Yaskawa INFORM job: Cilinder_ROBODK.jbi

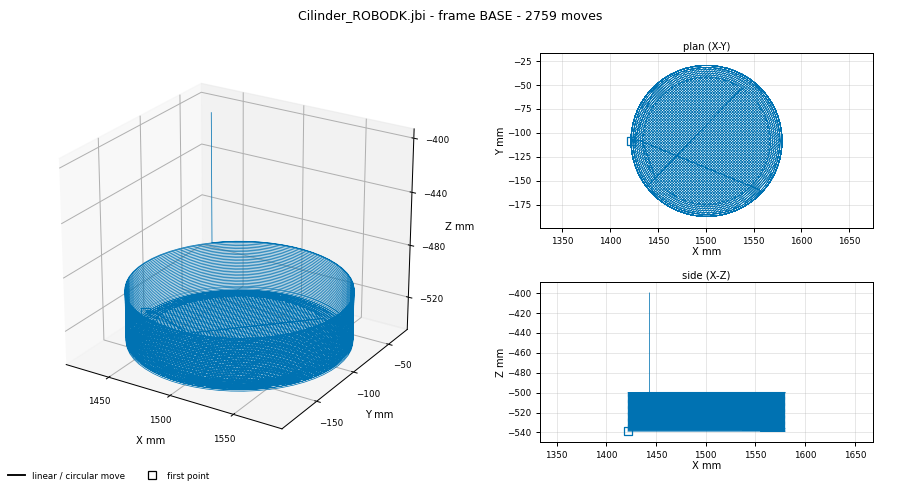
[picture p0: tool path of Cilinder_ROBODK.jbi in frame BASE, 2759 of 2760 moves have a stored position in this frame; points joined in program order, loops and branches not executed]
/JOB
//NAME CILINDER
//POS
///NPOS 2760,0,0,0,0,0
///TOOL 9
///POSTYPE PULSE
///PULSE
C00000=-4,42,-29,0,-18,-176
///TOOL 9
///POSTYPE BASE
///RECTAN
///RCONF 0,0,0,0,0,0,0,0
C00001=1421.799,-108.483,-538.800,180.00,-0.00,180.00
C00002=1422.262,-99.945,-538.800,180.00,0.00,-180.00
C00003=1423.646,-91.503,-538.800,180.00,-0.00,180.00
C00004=1425.931,-83.274,-538.800,180.00,-0.00,-180.00
C00005=1429.100,-75.315,-538.800,180.00,0.00,-180.00
C00006=1433.106,-67.758,-538.800,180.00,0.00,180.00
C00007=1437.906,-60.678,-538.800,180.00,-0.00,-180.00
C00008=1443.445,-54.158,-538.800,180.00,-0.00,-180.00
C00009=1449.655,-48.276,-538.800,180.00,0.00,180.00
C00010=1456.467,-43.098,-538.800,180.00,-0.00,-180.00
C00011=1463.794,-38.689,-538.800,180.00,-0.00,-180.00
C00012=1471.559,-35.097,-538.800,180.00,0.00,180.00
C00013=1479.661,-32.366,-538.800,180.00,0.00,-180.00
C00014=1488.017,-30.527,-538.800,180.00,0.00,180.00
C00015=1496.522,-29.601,-538.800,180.00,-0.00,180.00
C00016=1505.072,-29.601,-538.800,180.00,-0.00,-180.00
C00017=1513.577,-30.527,-538.800,180.00,-0.00,-180.00
C00018=1521.933,-32.366,-538.800,180.00,-0.00,-180.00
C00019=1530.035,-35.097,-538.800,180.00,0.00,180.00
C00020=1537.800,-38.689,-538.800,180.00,0.00,-180.00
C00021=1545.127,-43.098,-538.800,180.00,0.00,180.00
C00022=1551.939,-48.276,-538.800,180.00,0.00,-180.00
C00023=1558.149,-54.158,-538.800,180.00,0.00,-180.00
C00024=1563.688,-60.678,-538.800,180.00,-0.00,-180.00
C00025=1568.488,-67.758,-538.800,180.00,-0.00,180.00
C00026=1572.494,-75.315,-538.800,180.00,0.00,-180.00
C00027=1575.665,-83.274,-538.800,180.00,0.00,180.00
C00028=1577.948,-91.503,-538.800,180.00,0.00,-180.00
C00029=1579.332,-99.945,-538.800,180.00,-0.00,180.00
C00030=1579.795,-108.486,-538.800,180.00,0.00,-180.00
C00031=1579.332,-117.025,-538.800,180.00,0.00,-180.00
C00032=1577.948,-125.467,-538.800,180.00,-0.00,-180.00
C00033=1575.663,-133.694,-538.800,180.00,-0.00,-180.00
C00034=1572.494,-141.653,-538.800,180.00,-0.00,-180.00
C00035=1568.486,-149.212,-538.800,180.00,0.00,-180.00
C00036=1563.686,-156.292,-538.800,180.00,0.00,-180.00
C00037=1558.149,-162.810,-538.800,180.00,0.00,-180.00
C00038=1551.937,-168.694,-538.800,180.00,0.00,-180.00
C00039=1545.128,-173.870,-538.800,180.00,-0.00,-180.00
C00040=1537.800,-178.279,-538.800,180.00,-0.00,-180.00
C00041=1530.035,-181.871,-538.800,180.00,0.00,-180.00
C00042=1521.933,-184.602,-538.800,180.00,0.00,180.00
C00043=1513.577,-186.441,-538.800,180.00,0.00,-180.00
C00044=1505.072,-187.366,-538.800,180.00,0.00,-180.00
C00045=1496.522,-187.366,-538.800,180.00,0.00,180.00
C00046=1488.017,-186.441,-538.800,180.00,-0.00,-180.00
C00047=1479.661,-184.602,-538.800,180.00,-0.00,-180.00
C00048=1471.559,-181.871,-538.800,180.00,-0.00,-180.00
C00049=1463.794,-178.279,-538.800,180.00,-0.00,-180.00
C00050=1456.467,-173.870,-538.800,180.00,0.00,-180.00
C00051=1449.655,-168.692,-538.800,180.00,0.00,-180.00
C00052=1443.445,-162.810,-538.800,180.00,-0.00,-180.00
C00053=1437.906,-156.290,-538.800,180.00,0.00,-180.00
C00054=1433.106,-149.210,-538.800,180.00,0.00,-180.00
C00055=1429.100,-141.653,-538.800,180.00,0.00,180.00
C00056=1425.929,-133.694,-538.800,180.00,0.00,-180.00
C00057=1423.646,-125.465,-538.800,180.00,0.00,-180.00
C00058=1422.262,-117.023,-538.800,180.00,0.00,-180.00
C00059=1421.799,-108.483,-538.800,180.00,-0.00,180.00
C00060=1421.846,-107.610,-538.800,180.00,-0.00,-180.00
C00061=1424.567,-107.757,-538.800,180.00,0.00,-180.00
C00062=1424.528,-108.484,-538.800,180.00,-0.00,-180.00
C00063=1423.702,-108.482,-538.800,180.00,0.00,-180.00
C00064=1424.154,-100.153,-538.800,180.00,-0.00,180.00
C00065=1425.505,-91.912,-538.800,180.00,-0.00,-180.00
C00066=1427.735,-83.882,-538.800,180.00,0.00,-180.00
C00067=1430.827,-76.115,-538.800,180.00,0.00,-180.00
C00068=1434.736,-68.740,-538.800,180.00,-0.00,-180.00
C00069=1439.419,-61.831,-538.800,180.00,-0.00,-180.00
C00070=1444.826,-55.468,-538.800,180.00,0.00,-180.00
C00071=1450.887,-49.728,-538.800,180.00,-0.00,180.00
C00072=1457.537,-44.673,-538.800,180.00,0.00,-180.00
C00073=1464.686,-40.372,-538.800,180.00,-0.00,-180.00
C00074=1472.266,-36.865,-538.800,180.00,-0.00,-180.00
C00075=1480.169,-34.201,-538.800,180.00,0.00,-180.00
C00076=1488.326,-32.405,-538.800,180.00,0.00,-180.00
C00077=1496.627,-31.501,-538.800,180.00,-0.00,180.00
C00078=1504.967,-31.501,-538.800,180.00,0.00,-180.00
C00079=1513.268,-32.405,-538.800,180.00,0.00,-180.00
C00080=1521.425,-34.201,-538.800,180.00,0.00,-180.00
C00081=1529.328,-36.865,-538.800,180.00,-0.00,180.00
C00082=1536.908,-40.372,-538.800,180.00,-0.00,-180.00
C00083=1544.056,-44.673,-538.800,180.00,-0.00,180.00
C00084=1550.707,-49.728,-538.800,180.00,0.00,180.00
C00085=1556.768,-55.468,-538.800,180.00,0.00,-180.00
C00086=1562.175,-61.831,-538.800,180.00,-0.00,-180.00
C00087=1566.858,-68.740,-538.800,180.00,-0.00,-180.00
C00088=1570.767,-76.115,-538.800,180.00,-0.00,-180.00
C00089=1573.867,-83.896,-538.800,180.00,0.00,180.00
C00090=1576.089,-91.913,-538.800,180.00,-0.00,-180.00
C00091=1577.440,-100.153,-538.800,180.00,-0.00,-180.00
C00092=1577.892,-108.487,-538.800,180.00,0.00,-180.00
C00093=1577.440,-116.819,-538.800,180.00,-0.00,-180.00
C00094=1576.089,-125.059,-538.800,180.00,0.00,-180.00
C00095=1573.863,-133.072,-538.800,180.00,-0.00,180.00
C00096=1570.766,-140.853,-538.800,180.00,-0.00,-180.00
C00097=1566.854,-148.232,-538.800,180.00,-0.00,-180.00
C00098=1562.172,-155.139,-538.800,180.00,-0.00,-180.00
C00099=1556.768,-161.501,-538.800,180.00,0.00,-180.00
C00100=1550.703,-167.244,-538.800,180.00,-0.00,180.00
C00101=1544.058,-172.295,-538.800,180.00,-0.00,-180.00
C00102=1536.908,-176.596,-538.800,180.00,0.00,-180.00
C00103=1529.328,-180.103,-538.800,180.00,0.00,-180.00
C00104=1521.425,-182.767,-538.800,180.00,-0.00,180.00
C00105=1513.268,-184.563,-538.800,180.00,-0.00,-180.00
C00106=1504.967,-185.465,-538.800,180.00,-0.00,180.00
C00107=1496.627,-185.466,-538.800,180.00,-0.00,-180.00
C00108=1488.326,-184.563,-538.800,180.00,-0.00,180.00
C00109=1480.169,-182.767,-538.800,180.00,-0.00,-180.00
C00110=1472.266,-180.103,-538.800,180.00,0.00,-180.00
C00111=1464.686,-176.596,-538.800,180.00,0.00,-180.00
C00112=1457.537,-172.295,-538.800,180.00,0.00,-180.00
C00113=1450.887,-167.240,-538.800,180.00,0.00,180.00
C00114=1444.826,-161.500,-538.800,180.00,0.00,-180.00
C00115=1439.419,-155.137,-538.800,180.00,0.00,180.00
C00116=1434.736,-148.228,-538.800,180.00,0.00,-180.00
C00117=1430.827,-140.853,-538.800,180.00,0.00,180.00
C00118=1427.727,-133.072,-538.800,180.00,0.00,-180.00
C00119=1425.505,-125.055,-538.800,180.00,0.00,180.00
C00120=1424.154,-116.815,-538.800,180.00,0.00,-180.00
C00121=1423.702,-108.482,-538.800,180.00,0.00,-180.00
C00122=1424.528,-108.484,-538.800,180.00,-0.00,-180.00
C00123=1445.040,-56.761,-538.800,180.00,-0.00,180.00
C00124=1447.262,-54.539,-538.800,180.00,0.00,-180.00
C00125=1460.678,-43.951,-538.800,180.00,0.00,180.00
C00126=1436.060,-68.569,-538.800,180.00,-0.00,180.00
C00127=1435.707,-68.922,-538.800,180.00,0.00,-180.00
C00128=1432.654,-74.803,-538.800,180.00,0.00,-180.00
C00129=1467.099,-40.359,-538.800,180.00,0.00,-180.00
C00130=1467.452,-40.006,-538.800,180.00,-0.00,-180.00
C00131=1472.362,-37.924,-538.800,180.00,0.00,-180.00
C00132=1430.403,-79.883,-538.800,180.00,0.00,180.00
C00133=1430.050,-80.236,-538.800,180.00,-0.00,-180.00
C00134=1430.069,-80.243,-538.800,180.00,0.00,-180.00
C00135=1428.596,-84.518,-538.800,180.00,-0.00,-180.00
C00136=1476.681,-36.433,-538.800,180.00,0.00,180.00
C00137=1477.034,-36.080,-538.800,180.00,-0.00,-180.00
C00138=1477.047,-36.120,-538.800,180.00,-0.00,180.00
C00139=1480.871,-35.072,-538.800,180.00,0.00,-180.00
C00140=1427.508,-88.435,-538.800,180.00,0.00,-180.00
C00141=1427.155,-88.788,-538.800,180.00,0.00,-180.00
C00142=1427.222,-88.805,-538.800,180.00,0.00,-180.00
C00143=1426.450,-92.321,-538.800,180.00,-0.00,-180.00
C00144=1484.499,-34.273,-538.800,180.00,0.00,-180.00
C00145=1488.126,-33.474,-538.800,180.00,-0.00,180.00
C00146=1425.896,-95.704,-538.800,180.00,0.00,-180.00
C00147=1425.341,-99.087,-538.800,180.00,-0.00,180.00
C00148=1491.345,-33.083,-538.800,180.00,0.00,-180.00
C00149=1494.519,-32.738,-538.800,180.00,0.00,-180.00
C00150=1425.043,-102.214,-538.800,180.00,0.00,-180.00
C00151=1424.880,-105.205,-538.800,180.00,0.00,-180.00
C00152=1497.583,-32.502,-538.800,180.00,0.00,-180.00
C00153=1500.411,-32.502,-538.800,180.00,0.00,180.00
C00154=1424.718,-108.195,-538.800,180.00,0.00,-180.00
C00155=1424.834,-110.908,-538.800,180.00,0.00,180.00
C00156=1503.240,-32.502,-538.800,180.00,0.00,-180.00
C00157=1505.954,-32.616,-538.800,180.00,0.00,-180.00
C00158=1424.980,-113.590,-538.800,180.00,-0.00,180.00
C00159=1425.126,-116.273,-538.800,180.00,-0.00,-180.00
C00160=1508.505,-32.894,-538.800,180.00,0.00,180.00
C00161=1511.055,-33.172,-538.800,180.00,0.00,-180.00
C00162=1425.483,-118.744,-538.800,180.00,-0.00,180.00
C00163=1425.882,-121.174,-538.800,180.00,-0.00,-180.00
C00164=1513.561,-33.495,-538.800,180.00,-0.00,180.00
C00165=1515.879,-34.005,-538.800,180.00,-0.00,180.00
C00166=1426.280,-123.604,-538.800,180.00,0.00,-180.00
C00167=1426.784,-125.929,-538.800,180.00,-0.00,-180.00
C00168=1518.196,-34.516,-538.800,180.00,-0.00,180.00
C00169=1520.514,-35.027,-538.800,180.00,0.00,180.00
C00170=1427.398,-128.143,-538.800,180.00,-0.00,-180.00
C00171=1428.011,-130.358,-538.800,180.00,-0.00,180.00
C00172=1522.686,-35.683,-538.800,180.00,-0.00,180.00
C00173=1524.802,-36.396,-538.800,180.00,-0.00,180.00
C00174=1428.625,-132.573,-538.800,180.00,-0.00,-180.00
C00175=1429.415,-134.611,-538.800,180.00,0.00,-180.00
C00176=1526.917,-37.109,-538.800,180.00,-0.00,-180.00
C00177=1529.026,-37.829,-538.800,180.00,-0.00,180.00
C00178=1430.221,-136.634,-538.800,180.00,0.00,-180.00
C00179=1431.026,-138.657,-538.800,180.00,-0.00,180.00
C00180=1530.960,-38.723,-538.800,180.00,0.00,-180.00
C00181=1532.893,-39.619,-538.800,180.00,0.00,180.00
C00182=1431.853,-140.658,-538.800,180.00,-0.00,180.00
C00183=1432.833,-142.507,-538.800,180.00,0.00,180.00
C00184=1534.827,-40.513,-538.800,180.00,-0.00,-180.00
C00185=1536.733,-41.436,-538.800,180.00,0.00,-180.00
C00186=1433.812,-144.356,-538.800,180.00,-0.00,-180.00
C00187=1434.792,-146.204,-538.800,180.00,0.00,-180.00
C00188=1538.499,-42.498,-538.800,180.00,0.00,180.00
C00189=1540.265,-43.561,-538.800,180.00,0.00,-180.00
C00190=1435.802,-148.023,-538.800,180.00,0.00,-180.00
C00191=1436.945,-149.709,-538.800,180.00,0.00,-180.00
C00192=1542.030,-44.623,-538.800,180.00,0.00,-180.00
C00193=1543.769,-45.713,-538.800,180.00,0.00,180.00
C00194=1438.088,-151.394,-538.800,180.00,-0.00,-180.00
C00195=1439.230,-153.080,-538.800,180.00,0.00,-180.00
C00196=1545.376,-46.934,-538.800,180.00,-0.00,-180.00
C00197=1546.983,-48.155,-538.800,180.00,-0.00,-180.00
C00198=1440.395,-154.744,-538.800,180.00,0.00,-180.00
C00199=1441.695,-156.273,-538.800,180.00,0.00,-180.00
C00200=1548.590,-49.377,-538.800,180.00,-0.00,-180.00
C00201=1550.184,-50.612,-538.800,180.00,-0.00,180.00
C00202=1442.994,-157.802,-538.800,180.00,0.00,180.00
C00203=1444.293,-159.331,-538.800,180.00,0.00,-180.00
C00204=1551.636,-51.988,-538.800,180.00,0.00,-180.00
C00205=1553.089,-53.363,-538.800,180.00,-0.00,-180.00
C00206=1445.598,-160.855,-538.800,180.00,-0.00,-180.00
C00207=1447.051,-162.230,-538.800,180.00,-0.00,180.00
C00208=1554.542,-54.739,-538.800,180.00,0.00,180.00
C00209=1555.994,-56.115,-538.800,180.00,-0.00,-180.00
C00210=1448.503,-163.606,-538.800,180.00,0.00,-180.00
C00211=1449.956,-164.982,-538.800,180.00,0.00,-180.00
C00212=1557.299,-57.639,-538.800,180.00,0.00,-180.00
C00213=1558.598,-59.168,-538.800,180.00,-0.00,-180.00
C00214=1451.409,-166.357,-538.800,180.00,0.00,-180.00
C00215=1453.002,-167.593,-538.800,180.00,0.00,180.00
C00216=1559.898,-60.697,-538.800,180.00,-0.00,-180.00
C00217=1561.198,-62.225,-538.800,180.00,-0.00,-180.00
C00218=1454.609,-168.814,-538.800,180.00,0.00,-180.00
C00219=1456.216,-170.036,-538.800,180.00,0.00,-180.00
C00220=1562.362,-63.889,-538.800,180.00,0.00,-180.00
C00221=1563.504,-65.576,-538.800,180.00,-0.00,180.00
C00222=1457.823,-171.257,-538.800,180.00,-0.00,180.00
C00223=1459.562,-172.347,-538.800,180.00,-0.00,180.00
C00224=1564.647,-67.261,-538.800,180.00,0.00,-180.00
C00225=1565.790,-68.947,-538.800,180.00,-0.00,180.00
C00226=1461.328,-173.409,-538.800,180.00,-0.00,-180.00
C00227=1463.094,-174.472,-538.800,180.00,-0.00,180.00
C00228=1566.799,-70.766,-538.800,180.00,-0.00,-180.00
C00229=1567.779,-72.614,-538.800,180.00,0.00,180.00
C00230=1464.860,-175.534,-538.800,180.00,-0.00,180.00
C00231=1466.766,-176.456,-538.800,180.00,0.00,-180.00
C00232=1568.759,-74.463,-538.800,180.00,-0.00,-180.00
C00233=1569.739,-76.312,-538.800,180.00,-0.00,-180.00
C00234=1468.699,-177.352,-538.800,180.00,0.00,-180.00
C00235=1470.633,-178.246,-538.800,180.00,0.00,180.00
C00236=1570.565,-78.314,-538.800,180.00,0.00,-180.00
C00237=1571.372,-80.336,-538.800,180.00,-0.00,-180.00
C00238=1472.566,-179.141,-538.800,180.00,-0.00,-180.00
C00239=1474.675,-179.860,-538.800,180.00,0.00,-180.00
C00240=1572.178,-82.358,-538.800,180.00,0.00,180.00
C00241=1572.968,-84.397,-538.800,180.00,0.00,180.00
C00242=1476.791,-180.573,-538.800,180.00,-0.00,180.00
C00243=1478.906,-181.287,-538.800,180.00,0.00,-180.00
C00244=1573.581,-86.611,-538.800,180.00,0.00,-180.00
C00245=1574.195,-88.826,-538.800,180.00,0.00,-180.00
C00246=1481.078,-181.944,-538.800,180.00,0.00,-180.00
C00247=1483.395,-182.454,-538.800,180.00,-0.00,-180.00
C00248=1574.809,-91.041,-538.800,180.00,-0.00,-180.00
C00249=1575.313,-93.365,-538.800,180.00,0.00,-180.00
C00250=1485.713,-182.965,-538.800,180.00,0.00,-180.00
C00251=1488.031,-183.475,-538.800,180.00,0.00,-180.00
C00252=1575.711,-95.795,-538.800,180.00,0.00,-180.00
C00253=1576.109,-98.226,-538.800,180.00,-0.00,180.00
C00254=1490.537,-183.798,-538.800,180.00,-0.00,-180.00
C00255=1493.088,-184.075,-538.800,180.00,0.00,180.00
C00256=1576.466,-100.697,-538.800,180.00,-0.00,180.00
C00257=1576.612,-103.380,-538.800,180.00,0.00,-180.00
C00258=1495.639,-184.353,-538.800,180.00,-0.00,-180.00
C00259=1498.354,-184.466,-538.800,180.00,0.00,180.00
C00260=1576.758,-106.062,-538.800,180.00,0.00,180.00
C00261=1576.874,-108.774,-538.800,180.00,0.00,-180.00
C00262=1501.183,-184.466,-538.800,180.00,0.00,180.00
C00263=1504.011,-184.466,-538.800,180.00,0.00,-180.00
C00264=1576.712,-111.765,-538.800,180.00,-0.00,-180.00
C00265=1576.549,-114.756,-538.800,180.00,0.00,-180.00
C00266=1507.075,-184.230,-538.800,180.00,-0.00,180.00
C00267=1510.248,-183.886,-538.800,180.00,0.00,-180.00
C00268=1576.251,-117.883,-538.800,180.00,0.00,180.00
C00269=1575.696,-121.266,-538.800,180.00,-0.00,-180.00
C00270=1513.467,-183.496,-538.800,180.00,-0.00,-180.00
C00271=1517.093,-182.697,-538.800,180.00,0.00,180.00
C00272=1575.143,-124.648,-538.800,180.00,0.00,-180.00
C00273=1575.496,-124.295,-538.800,180.00,0.00,-180.00
C00274=1575.383,-124.277,-538.800,180.00,-0.00,180.00
C00275=1574.085,-128.534,-538.800,180.00,0.00,-180.00
C00276=1520.721,-181.898,-538.800,180.00,-0.00,180.00
C00277=1520.368,-182.251,-538.800,180.00,0.00,-180.00
C00278=1520.348,-182.163,-538.800,180.00,-0.00,-180.00
C00279=1524.911,-180.536,-538.800,180.00,-0.00,-180.00
C00280=1572.997,-132.450,-538.800,180.00,0.00,180.00
C00281=1573.350,-132.097,-538.800,180.00,0.00,-180.00
C00282=1573.284,-132.080,-538.800,180.00,0.00,-180.00
C00283=1571.188,-137.088,-538.800,180.00,0.00,-180.00
C00284=1529.230,-179.046,-538.800,180.00,-0.00,180.00
C00285=1528.877,-179.399,-538.800,180.00,0.00,-180.00
C00286=1528.874,-179.390,-538.800,180.00,-0.00,-180.00
C00287=1534.493,-176.611,-538.800,180.00,-0.00,180.00
C00288=1568.937,-142.167,-538.800,180.00,0.00,-180.00
C00289=1569.290,-141.814,-538.800,180.00,0.00,-180.00
C00290=1565.528,-148.405,-538.800,180.00,0.00,-180.00
C00291=1540.914,-173.018,-538.800,180.00,-0.00,180.00
C00292=1540.561,-173.371,-538.800,180.00,-0.00,-180.00
C00293=1554.330,-162.432,-538.800,180.00,0.00,-180.00
C00294=1556.551,-160.211,-538.800,180.00,-0.00,180.00
C00295=1555.237,-159.097,-538.800,180.00,0.00,180.00
C00296=1555.237,-159.097,-537.600,180.00,0.00,180.00
C00297=1431.814,-108.483,-537.600,180.00,-0.00,180.00
C00298=1432.218,-101.027,-537.600,180.00,0.00,-180.00
C00299=1433.426,-93.656,-537.600,180.00,-0.00,-180.00
C00300=1435.421,-86.471,-537.600,180.00,-0.00,-180.00
C00301=1438.190,-79.519,-537.600,180.00,0.00,-180.00
C00302=1441.687,-72.920,-537.600,180.00,0.00,180.00
C00303=1445.878,-66.739,-537.600,180.00,-0.00,-180.00
C00304=1450.715,-61.046,-537.600,180.00,-0.00,180.00
C00305=1456.138,-55.909,-537.600,180.00,0.00,-180.00
C00306=1462.087,-51.388,-537.600,180.00,0.00,-180.00
C00307=1468.485,-47.537,-537.600,180.00,0.00,-180.00
C00308=1475.266,-44.400,-537.600,180.00,0.00,-180.00
C00309=1482.341,-42.016,-537.600,180.00,-0.00,180.00
C00310=1489.637,-40.409,-537.600,180.00,0.00,-180.00
C00311=1497.064,-39.601,-537.600,180.00,-0.00,-180.00
C00312=1504.530,-39.601,-537.600,180.00,0.00,-180.00
C00313=1511.957,-40.409,-537.600,180.00,0.00,-180.00
C00314=1519.253,-42.016,-537.600,180.00,0.00,-180.00
C00315=1526.328,-44.400,-537.600,180.00,-0.00,180.00
C00316=1533.109,-47.537,-537.600,180.00,0.00,-180.00
C00317=1539.507,-51.387,-537.600,180.00,-0.00,180.00
C00318=1545.456,-55.909,-537.600,180.00,0.00,-180.00
C00319=1550.879,-61.046,-537.600,180.00,0.00,-180.00
C00320=1555.716,-66.739,-537.600,180.00,0.00,180.00
C00321=1559.907,-72.920,-537.600,180.00,0.00,180.00
C00322=1563.404,-79.520,-537.600,180.00,-0.00,-180.00
C00323=1566.175,-86.471,-537.600,180.00,-0.00,-180.00
C00324=1568.167,-93.654,-537.600,180.00,0.00,180.00
C00325=1569.376,-101.027,-537.600,180.00,0.00,180.00
C00326=1569.780,-108.486,-537.600,180.00,-0.00,180.00
C00327=1569.376,-115.943,-537.600,180.00,-0.00,-180.00
C00328=1568.168,-123.314,-537.600,180.00,0.00,-180.00
C00329=1566.173,-130.496,-537.600,180.00,0.00,180.00
C00330=1563.404,-137.449,-537.600,180.00,0.00,180.00
C00331=1559.905,-144.049,-537.600,180.00,0.00,180.00
C00332=1555.714,-150.232,-537.600,180.00,-0.00,-180.00
C00333=1550.879,-155.922,-537.600,180.00,-0.00,-180.00
C00334=1545.454,-161.061,-537.600,180.00,-0.00,-180.00
C00335=1539.508,-165.580,-537.600,180.00,-0.00,-180.00
C00336=1533.109,-169.430,-537.600,180.00,0.00,-180.00
C00337=1526.328,-172.568,-537.600,180.00,-0.00,180.00
C00338=1519.253,-174.952,-537.600,180.00,-0.00,-180.00
C00339=1511.957,-176.558,-537.600,180.00,0.00,-180.00
C00340=1504.530,-177.366,-537.600,180.00,0.00,-180.00
C00341=1497.064,-177.366,-537.600,180.00,0.00,180.00
C00342=1489.637,-176.558,-537.600,180.00,-0.00,180.00
C00343=1482.341,-174.952,-537.600,180.00,-0.00,-180.00
C00344=1475.266,-172.568,-537.600,180.00,0.00,-180.00
C00345=1468.485,-169.431,-537.600,180.00,0.00,180.00
C00346=1462.087,-165.581,-537.600,180.00,0.00,180.00
C00347=1456.138,-161.059,-537.600,180.00,-0.00,-180.00
C00348=1450.715,-155.922,-537.600,180.00,-0.00,180.00
C00349=1445.878,-150.229,-537.600,180.00,0.00,180.00
C00350=1441.687,-144.048,-537.600,180.00,0.00,-180.00
C00351=1438.190,-137.448,-537.600,180.00,0.00,-180.00
C00352=1435.419,-130.497,-537.600,180.00,-0.00,-180.00
C00353=1433.426,-123.314,-537.600,180.00,-0.00,-180.00
C00354=1432.218,-115.941,-537.600,180.00,-0.00,180.00
C00355=1431.814,-108.483,-537.600,180.00,-0.00,180.00
C00356=1429.811,-108.483,-537.600,180.00,-0.00,-180.00
C00357=1430.227,-100.811,-537.600,180.00,-0.00,-180.00
C00358=1431.470,-93.225,-537.600,180.00,-0.00,-180.00
C00359=1433.523,-85.832,-537.600,180.00,-0.00,-180.00
C00360=1436.372,-78.678,-537.600,180.00,0.00,-180.00
C00361=1439.971,-71.888,-537.600,180.00,0.00,-180.00
C00362=1444.284,-65.526,-537.600,180.00,0.00,-180.00
C00363=1449.261,-59.668,-537.600,180.00,-0.00,-180.00
C00364=1454.841,-54.382,-537.600,180.00,0.00,180.00
C00365=1460.963,-49.730,-537.600,180.00,-0.00,180.00
C00366=1467.547,-45.768,-537.600,180.00,0.00,-180.00
C00367=1474.525,-42.540,-537.600,180.00,-0.00,-180.00
C00368=1481.805,-40.086,-537.600,180.00,0.00,-180.00
C00369=1489.313,-38.433,-537.600,180.00,-0.00,-180.00
C00370=1496.956,-37.601,-537.600,180.00,0.00,-180.00
C00371=1504.638,-37.601,-537.600,180.00,-0.00,180.00
C00372=1512.281,-38.433,-537.600,180.00,0.00,-180.00
C00373=1519.789,-40.086,-537.600,180.00,0.00,180.00
C00374=1527.069,-42.540,-537.600,180.00,-0.00,-180.00
C00375=1534.047,-45.768,-537.600,180.00,0.00,180.00
C00376=1540.631,-49.730,-537.600,180.00,-0.00,180.00
C00377=1546.753,-54.382,-537.600,180.00,-0.00,-180.00
C00378=1552.333,-59.668,-537.600,180.00,-0.00,-180.00
C00379=1557.310,-65.526,-537.600,180.00,-0.00,180.00
C00380=1561.623,-71.888,-537.600,180.00,0.00,-180.00
C00381=1565.222,-78.679,-537.600,180.00,-0.00,-180.00
C00382=1568.073,-85.832,-537.600,180.00,0.00,-180.00
C00383=1570.124,-93.224,-537.600,180.00,0.00,180.00
C00384=1571.367,-100.811,-537.600,180.00,0.00,-180.00
C00385=1571.783,-108.486,-537.600,180.00,0.00,-180.00
C00386=1571.367,-116.159,-537.600,180.00,-0.00,-180.00
C00387=1570.124,-123.745,-537.600,180.00,-0.00,-180.00
C00388=1568.071,-131.136,-537.600,180.00,0.00,-180.00
C00389=1565.222,-138.290,-537.600,180.00,-0.00,-180.00
C00390=1561.621,-145.082,-537.600,180.00,-0.00,-180.00
C00391=1557.308,-151.444,-537.600,180.00,-0.00,180.00
C00392=1552.333,-157.300,-537.600,180.00,0.00,180.00
C00393=1546.751,-162.588,-537.600,180.00,0.00,-180.00
C00394=1540.632,-167.238,-537.600,180.00,0.00,-180.00
C00395=1534.048,-171.200,-537.600,180.00,-0.00,-180.00
C00396=1527.069,-174.428,-537.600,180.00,0.00,180.00
C00397=1519.789,-176.882,-537.600,180.00,0.00,180.00
C00398=1512.281,-178.535,-537.600,180.00,0.00,-180.00
C00399=1504.638,-179.366,-537.600,180.00,0.00,-180.00
C00400=1496.956,-179.366,-537.600,180.00,-0.00,180.00
C00401=1489.313,-178.535,-537.600,180.00,-0.00,-180.00
C00402=1481.805,-176.882,-537.600,180.00,0.00,180.00
C00403=1474.525,-174.428,-537.600,180.00,0.00,-180.00
C00404=1467.547,-171.200,-537.600,180.00,0.00,-180.00
C00405=1460.963,-167.238,-537.600,180.00,0.00,180.00
C00406=1454.841,-162.586,-537.600,180.00,-0.00,-180.00
C00407=1449.261,-157.300,-537.600,180.00,-0.00,180.00
C00408=1444.284,-151.442,-537.600,180.00,0.00,-180.00
C00409=1439.971,-145.080,-537.600,180.00,-0.00,-180.00
C00410=1436.372,-138.289,-537.600,180.00,0.00,-180.00
C00411=1433.521,-131.136,-537.600,180.00,-0.00,-180.00
C00412=1431.470,-123.744,-537.600,180.00,0.00,-180.00
C00413=1430.227,-116.157,-537.600,180.00,0.00,-180.00
C00414=1429.811,-108.483,-537.600,180.00,-0.00,-180.00
C00415=1427.808,-108.483,-537.600,180.00,-0.00,-180.00
C00416=1428.236,-100.594,-537.600,180.00,0.00,180.00
C00417=1429.514,-92.794,-537.600,180.00,-0.00,-180.00
C00418=1431.625,-85.192,-537.600,180.00,-0.00,-180.00
C00419=1434.554,-77.837,-537.600,180.00,0.00,-180.00
C00420=1438.255,-70.855,-537.600,180.00,-0.00,180.00
C00421=1442.689,-64.314,-537.600,180.00,-0.00,-180.00
C00422=1447.807,-58.291,-537.600,180.00,0.00,180.00
C00423=1453.545,-52.856,-537.600,180.00,0.00,180.00
C00424=1459.839,-48.072,-537.600,180.00,-0.00,180.00
C00425=1466.608,-43.998,-537.600,180.00,0.00,-180.00
C00426=1473.783,-40.679,-537.600,180.00,0.00,-180.00
C00427=1481.269,-38.156,-537.600,180.00,-0.00,-180.00
C00428=1488.989,-36.456,-537.600,180.00,0.00,-180.00
C00429=1496.847,-35.601,-537.600,180.00,0.00,180.00
C00430=1504.747,-35.601,-537.600,180.00,-0.00,180.00
C00431=1512.605,-36.456,-537.600,180.00,-0.00,-180.00
C00432=1520.325,-38.156,-537.600,180.00,-0.00,-180.00
C00433=1527.811,-40.679,-537.600,180.00,0.00,-180.00
C00434=1534.986,-43.998,-537.600,180.00,0.00,-180.00
C00435=1541.755,-48.072,-537.600,180.00,-0.00,180.00
C00436=1548.049,-52.856,-537.600,180.00,-0.00,-180.00
C00437=1553.787,-58.291,-537.600,180.00,0.00,-180.00
C00438=1558.905,-64.314,-537.600,180.00,-0.00,-180.00
C00439=1563.339,-70.855,-537.600,180.00,0.00,-180.00
C00440=1567.040,-77.838,-537.600,180.00,0.00,180.00
C00441=1569.971,-85.193,-537.600,180.00,0.00,180.00
C00442=1572.080,-92.794,-537.600,180.00,-0.00,-180.00
C00443=1573.358,-100.594,-537.600,180.00,0.00,-180.00
C00444=1573.786,-108.486,-537.600,180.00,0.00,-180.00
C00445=1573.358,-116.376,-537.600,180.00,0.00,180.00
C00446=1572.080,-124.175,-537.600,180.00,-0.00,180.00
C00447=1569.969,-131.775,-537.600,180.00,0.00,-180.00
C00448=1567.040,-139.131,-537.600,180.00,0.00,180.00
C00449=1563.338,-146.114,-537.600,180.00,-0.00,-180.00
C00450=1558.903,-152.656,-537.600,180.00,0.00,180.00
C00451=1553.787,-158.677,-537.600,180.00,0.00,-180.00
C00452=1548.047,-164.114,-537.600,180.00,0.00,180.00
C00453=1541.756,-168.896,-537.600,180.00,0.00,-180.00
C00454=1534.986,-172.970,-537.600,180.00,0.00,-180.00
C00455=1527.811,-176.289,-537.600,180.00,-0.00,-180.00
C00456=1520.325,-178.812,-537.600,180.00,0.00,-180.00
C00457=1512.605,-180.512,-537.600,180.00,-0.00,-180.00
C00458=1504.747,-181.366,-537.600,180.00,0.00,-180.00
C00459=1496.847,-181.366,-537.600,180.00,0.00,-180.00
C00460=1488.989,-180.512,-537.600,180.00,-0.00,180.00
C00461=1481.269,-178.812,-537.600,180.00,-0.00,180.00
C00462=1473.783,-176.289,-537.600,180.00,-0.00,180.00
C00463=1466.608,-172.970,-537.600,180.00,0.00,-180.00
C00464=1459.839,-168.896,-537.600,180.00,0.00,-180.00
C00465=1453.545,-164.112,-537.600,180.00,-0.00,-180.00
C00466=1447.807,-158.677,-537.600,180.00,0.00,-180.00
C00467=1442.689,-152.654,-537.600,180.00,0.00,-180.00
C00468=1438.255,-146.113,-537.600,180.00,-0.00,-180.00
C00469=1434.554,-139.130,-537.600,180.00,0.00,-180.00
C00470=1431.623,-131.776,-537.600,180.00,-0.00,180.00
C00471=1429.514,-124.174,-537.600,180.00,0.00,-180.00
C00472=1428.236,-116.374,-537.600,180.00,0.00,-180.00
C00473=1427.808,-108.483,-537.600,180.00,-0.00,-180.00
C00474=1425.805,-108.483,-537.600,180.00,-0.00,180.00
C00475=1426.245,-100.378,-537.600,180.00,-0.00,-180.00
C00476=1427.558,-92.364,-537.600,180.00,0.00,-180.00
C00477=1429.727,-84.553,-537.600,180.00,-0.00,-180.00
C00478=1432.736,-76.996,-537.600,180.00,0.00,-180.00
C00479=1436.538,-69.823,-537.600,180.00,0.00,-180.00
C00480=1441.095,-63.102,-537.600,180.00,0.00,-180.00
C00481=1446.353,-56.913,-537.600,180.00,0.00,-180.00
C00482=1452.248,-51.329,-537.600,180.00,0.00,-180.00
C00483=1458.715,-46.414,-537.600,180.00,-0.00,-180.00
C00484=1465.670,-42.229,-537.600,180.00,-0.00,-180.00
C00485=1473.042,-38.818,-537.600,180.00,0.00,-180.00
C00486=1480.733,-36.226,-537.600,180.00,-0.00,-180.00
C00487=1488.665,-34.480,-537.600,180.00,0.00,180.00
C00488=1496.739,-33.601,-537.600,180.00,0.00,-180.00
C00489=1504.855,-33.601,-537.600,180.00,0.00,180.00
C00490=1512.929,-34.480,-537.600,180.00,-0.00,-180.00
C00491=1520.861,-36.226,-537.600,180.00,-0.00,180.00
C00492=1528.552,-38.818,-537.600,180.00,-0.00,-180.00
C00493=1535.924,-42.229,-537.600,180.00,0.00,-180.00
C00494=1542.879,-46.414,-537.600,180.00,0.00,180.00
C00495=1549.346,-51.329,-537.600,180.00,-0.00,180.00
C00496=1555.241,-56.913,-537.600,180.00,0.00,180.00
C00497=1560.499,-63.102,-537.600,180.00,0.00,-180.00
C00498=1565.056,-69.823,-537.600,180.00,-0.00,-180.00
C00499=1568.858,-76.997,-537.600,180.00,-0.00,-180.00
C00500=1571.869,-84.553,-537.600,180.00,-0.00,180.00
C00501=1574.036,-92.363,-537.600,180.00,-0.00,180.00
C00502=1575.349,-100.378,-537.600,180.00,-0.00,-180.00
C00503=1575.789,-108.486,-537.600,180.00,-0.00,180.00
C00504=1575.350,-116.592,-537.600,180.00,0.00,180.00
C00505=1574.036,-124.606,-537.600,180.00,0.00,-180.00
C00506=1571.867,-132.415,-537.600,180.00,-0.00,-180.00
C00507=1568.858,-139.971,-537.600,180.00,-0.00,180.00
C00508=1565.054,-147.147,-537.600,180.00,0.00,-180.00
C00509=1560.497,-153.868,-537.600,180.00,0.00,180.00
C00510=1555.241,-160.055,-537.600,180.00,0.00,-180.00
C00511=1549.344,-165.641,-537.600,180.00,0.00,-180.00
C00512=1542.880,-170.554,-537.600,180.00,0.00,-180.00
C00513=1535.924,-174.739,-537.600,180.00,-0.00,-180.00
C00514=1528.552,-178.150,-537.600,180.00,0.00,-180.00
C00515=1520.861,-180.742,-537.600,180.00,-0.00,-180.00
C00516=1512.929,-182.488,-537.600,180.00,0.00,-180.00
C00517=1504.855,-183.366,-537.600,180.00,0.00,-180.00
C00518=1496.739,-183.366,-537.600,180.00,-0.00,-180.00
C00519=1488.665,-182.488,-537.600,180.00,0.00,-180.00
C00520=1480.733,-180.742,-537.600,180.00,0.00,-180.00
C00521=1473.042,-178.150,-537.600,180.00,-0.00,-180.00
C00522=1465.670,-174.739,-537.600,180.00,0.00,-180.00
C00523=1458.715,-170.554,-537.600,180.00,-0.00,-180.00
C00524=1452.248,-165.639,-537.600,180.00,0.00,-180.00
C00525=1446.353,-160.055,-537.600,180.00,0.00,-180.00
C00526=1441.095,-153.866,-537.600,180.00,0.00,180.00
C00527=1436.538,-147.145,-537.600,180.00,-0.00,-180.00
C00528=1432.736,-139.971,-537.600,180.00,0.00,-180.00
C00529=1429.725,-132.415,-537.600,180.00,-0.00,-180.00
C00530=1427.558,-124.605,-537.600,180.00,-0.00,-180.00
C00531=1426.245,-116.590,-537.600,180.00,-0.00,-180.00
C00532=1425.805,-108.483,-537.600,180.00,-0.00,180.00
C00533=1424.528,-108.484,-537.600,180.00,0.00,-180.00
C00534=1423.802,-108.483,-537.600,180.00,-0.00,180.00
C00535=1424.253,-100.161,-537.600,180.00,-0.00,180.00
C00536=1425.602,-91.933,-537.600,180.00,0.00,180.00
C00537=1427.829,-83.914,-537.600,180.00,0.00,180.00
C00538=1430.918,-76.156,-537.600,180.00,-0.00,-180.00
C00539=1434.822,-68.790,-537.600,180.00,-0.00,-180.00
C00540=1439.500,-61.890,-537.600,180.00,0.00,180.00
C00541=1444.899,-55.536,-537.600,180.00,-0.00,-180.00
C00542=1450.951,-49.802,-537.600,180.00,0.00,-180.00
C00543=1457.591,-44.756,-537.600,180.00,-0.00,180.00
C00544=1464.732,-40.459,-537.600,180.00,0.00,-180.00
C00545=1472.301,-36.958,-537.600,180.00,0.00,-180.00
C00546=1480.197,-34.296,-537.600,180.00,-0.00,180.00
C00547=1488.341,-32.503,-537.600,180.00,-0.00,-180.00
C00548=1496.630,-31.601,-537.600,180.00,-0.00,-180.00
C00549=1504.964,-31.601,-537.600,180.00,-0.00,180.00
C00550=1513.253,-32.503,-537.600,180.00,0.00,-180.00
C00551=1521.397,-34.296,-537.600,180.00,0.00,-180.00
C00552=1529.293,-36.958,-537.600,180.00,-0.00,-180.00
C00553=1536.862,-40.459,-537.600,180.00,0.00,180.00
C00554=1544.003,-44.756,-537.600,180.00,-0.00,-180.00
C00555=1550.643,-49.802,-537.600,180.00,-0.00,-180.00
C00556=1556.695,-55.536,-537.600,180.00,-0.00,-180.00
C00557=1562.094,-61.890,-537.600,180.00,0.00,-180.00
C00558=1566.772,-68.790,-537.600,180.00,0.00,-180.00
C00559=1570.676,-76.156,-537.600,180.00,0.00,-180.00
C00560=1573.767,-83.914,-537.600,180.00,0.00,-180.00
C00561=1575.992,-91.933,-537.600,180.00,0.00,-180.00
C00562=1577.341,-100.161,-537.600,180.00,0.00,-180.00
C00563=1577.792,-108.486,-537.600,180.00,0.00,-180.00
C00564=1577.341,-116.809,-537.600,180.00,0.00,-180.00
C00565=1575.992,-125.037,-537.600,180.00,0.00,-180.00
C00566=1573.765,-133.054,-537.600,180.00,0.00,180.00
C00567=1570.676,-140.812,-537.600,180.00,0.00,-180.00
C00568=1566.770,-148.180,-537.600,180.00,0.00,180.00
C00569=1562.092,-155.080,-537.600,180.00,0.00,180.00
C00570=1556.695,-161.432,-537.600,180.00,-0.00,-180.00
C00571=1550.641,-167.168,-537.600,180.00,0.00,-180.00
C00572=1544.004,-172.212,-537.600,180.00,0.00,-180.00
C00573=1536.862,-176.509,-537.600,180.00,0.00,-180.00
C00574=1529.293,-180.010,-537.600,180.00,0.00,180.00
C00575=1521.397,-182.672,-537.600,180.00,0.00,-180.00
C00576=1513.253,-184.465,-537.600,180.00,0.00,-180.00
C00577=1504.964,-185.366,-537.600,180.00,0.00,-180.00
C00578=1496.630,-185.366,-537.600,180.00,-0.00,-180.00
C00579=1488.341,-184.465,-537.600,180.00,0.00,-180.00
C00580=1480.197,-182.672,-537.600,180.00,-0.00,-180.00
C00581=1472.301,-180.010,-537.600,180.00,0.00,-180.00
C00582=1464.732,-176.509,-537.600,180.00,0.00,180.00
C00583=1457.591,-172.212,-537.600,180.00,0.00,-180.00
C00584=1450.951,-167.166,-537.600,180.00,0.00,180.00
C00585=1444.899,-161.432,-537.600,180.00,-0.00,-180.00
C00586=1439.500,-155.078,-537.600,180.00,-0.00,-180.00
C00587=1434.822,-148.178,-537.600,180.00,-0.00,-180.00
C00588=1430.918,-140.812,-537.600,180.00,0.00,-180.00
C00589=1427.827,-133.054,-537.600,180.00,-0.00,-180.00
C00590=1425.602,-125.035,-537.600,180.00,0.00,180.00
C00591=1424.253,-116.807,-537.600,180.00,0.00,-180.00
C00592=1423.802,-108.483,-537.600,180.00,-0.00,180.00
C00593=1424.528,-108.484,-537.600,180.00,0.00,-180.00
C00594=1421.799,-108.483,-537.600,180.00,0.00,180.00
C00595=1422.262,-99.945,-537.600,180.00,0.00,-180.00
C00596=1423.646,-91.503,-537.600,180.00,-0.00,-180.00
C00597=1425.931,-83.274,-537.600,180.00,-0.00,-180.00
C00598=1429.100,-75.315,-537.600,180.00,-0.00,-180.00
C00599=1433.106,-67.758,-537.600,180.00,-0.00,180.00
C00600=1437.906,-60.678,-537.600,180.00,-0.00,-180.00
C00601=1443.445,-54.158,-537.600,180.00,0.00,-180.00
C00602=1449.655,-48.276,-537.600,180.00,0.00,180.00
C00603=1456.467,-43.098,-537.600,180.00,0.00,-180.00
C00604=1463.794,-38.689,-537.600,180.00,0.00,-180.00
C00605=1471.559,-35.097,-537.600,180.00,-0.00,180.00
C00606=1479.661,-32.366,-537.600,180.00,-0.00,-180.00
C00607=1488.017,-30.527,-537.600,180.00,0.00,180.00
C00608=1496.522,-29.601,-537.600,180.00,0.00,180.00
C00609=1505.072,-29.601,-537.600,180.00,0.00,-180.00
C00610=1513.577,-30.527,-537.600,180.00,0.00,-180.00
C00611=1521.933,-32.366,-537.600,180.00,0.00,-180.00
C00612=1530.035,-35.097,-537.600,180.00,0.00,180.00
C00613=1537.800,-38.689,-537.600,180.00,0.00,-180.00
C00614=1545.127,-43.098,-537.600,180.00,0.00,180.00
C00615=1551.939,-48.276,-537.600,180.00,-0.00,-180.00
C00616=1558.149,-54.158,-537.600,180.00,0.00,-180.00
C00617=1563.688,-60.678,-537.600,180.00,0.00,180.00
C00618=1568.488,-67.758,-537.600,180.00,-0.00,180.00
C00619=1572.494,-75.315,-537.600,180.00,0.00,-180.00
C00620=1575.665,-83.274,-537.600,180.00,0.00,180.00
C00621=1577.948,-91.503,-537.600,180.00,-0.00,-180.00
C00622=1579.332,-99.945,-537.600,180.00,0.00,180.00
C00623=1579.795,-108.486,-537.600,180.00,0.00,-180.00
C00624=1579.332,-117.025,-537.600,180.00,-0.00,-180.00
C00625=1577.948,-125.467,-537.600,180.00,-0.00,-180.00
C00626=1575.663,-133.694,-537.600,180.00,-0.00,-180.00
C00627=1572.494,-141.653,-537.600,180.00,-0.00,-180.00
C00628=1568.486,-149.212,-537.600,180.00,-0.00,-180.00
C00629=1563.686,-156.292,-537.600,180.00,0.00,-180.00
C00630=1558.149,-162.810,-537.600,180.00,0.00,-180.00
C00631=1551.937,-168.694,-537.600,180.00,-0.00,-180.00
C00632=1545.128,-173.870,-537.600,180.00,-0.00,-180.00
C00633=1537.800,-178.279,-537.600,180.00,-0.00,-180.00
C00634=1530.035,-181.871,-537.600,180.00,0.00,-180.00
C00635=1521.933,-184.602,-537.600,180.00,-0.00,180.00
C00636=1513.577,-186.441,-537.600,180.00,0.00,-180.00
C00637=1505.072,-187.366,-537.600,180.00,0.00,-180.00
C00638=1496.522,-187.366,-537.600,180.00,-0.00,180.00
C00639=1488.017,-186.441,-537.600,180.00,0.00,-180.00
C00640=1479.661,-184.602,-537.600,180.00,-0.00,-180.00
C00641=1471.559,-181.871,-537.600,180.00,-0.00,-180.00
C00642=1463.794,-178.279,-537.600,180.00,0.00,-180.00
C00643=1456.467,-173.870,-537.600,180.00,0.00,-180.00
C00644=1449.655,-168.692,-537.600,180.00,-0.00,-180.00
C00645=1443.445,-162.810,-537.600,180.00,0.00,-180.00
C00646=1437.906,-156.290,-537.600,180.00,0.00,-180.00
C00647=1433.106,-149.210,-537.600,180.00,0.00,-180.00
C00648=1429.100,-141.653,-537.600,180.00,-0.00,180.00
C00649=1425.929,-133.694,-537.600,180.00,0.00,-180.00
C00650=1423.646,-125.465,-537.600,180.00,-0.00,-180.00
C00651=1422.262,-117.023,-537.600,180.00,0.00,180.00
C00652=1421.799,-108.483,-537.600,180.00,0.00,180.00
C00653=1421.846,-107.610,-537.600,180.00,0.00,-180.00
C00654=1424.567,-107.757,-537.600,180.00,0.00,-180.00
C00655=1433.717,-108.482,-537.600,180.00,-0.00,-180.00
C00656=1434.110,-101.236,-537.600,180.00,0.00,180.00
C00657=1435.285,-94.065,-537.600,180.00,-0.00,-180.00
C00658=1437.225,-87.079,-537.600,180.00,0.00,180.00
C00659=1439.917,-80.319,-537.600,180.00,-0.00,-180.00
C00660=1443.318,-73.902,-537.600,180.00,0.00,-180.00
C00661=1447.392,-67.892,-537.600,180.00,0.00,-180.00
C00662=1452.096,-62.356,-537.600,180.00,0.00,-180.00
C00663=1457.370,-57.361,-537.600,180.00,-0.00,-180.00
C00664=1463.157,-52.962,-537.600,180.00,0.00,180.00
C00665=1469.377,-49.220,-537.600,180.00,0.00,180.00
C00666=1475.973,-46.169,-537.600,180.00,-0.00,180.00
C00667=1482.849,-43.851,-537.600,180.00,0.00,-180.00
C00668=1489.946,-42.288,-537.600,180.00,0.00,180.00
C00669=1497.169,-41.501,-537.600,180.00,-0.00,-180.00
C00670=1504.425,-41.501,-537.600,180.00,-0.00,-180.00
C00671=1511.648,-42.288,-537.600,180.00,0.00,-180.00
C00672=1518.745,-43.851,-537.600,180.00,0.00,180.00
C00673=1525.621,-46.169,-537.600,180.00,0.00,180.00
C00674=1532.217,-49.220,-537.600,180.00,0.00,-180.00
C00675=1538.437,-52.962,-537.600,180.00,0.00,-180.00
C00676=1544.224,-57.361,-537.600,180.00,-0.00,-180.00
C00677=1549.498,-62.356,-537.600,180.00,-0.00,-180.00
C00678=1554.203,-67.892,-537.600,180.00,-0.00,-180.00
C00679=1558.277,-73.902,-537.600,180.00,0.00,180.00
C00680=1561.677,-80.320,-537.600,180.00,0.00,-180.00
C00681=1564.376,-87.093,-537.600,180.00,-0.00,-180.00
C00682=1566.308,-94.064,-537.600,180.00,0.00,180.00
C00683=1567.484,-101.235,-537.600,180.00,-0.00,-180.00
C00684=1567.877,-108.487,-537.600,180.00,0.00,180.00
C00685=1567.484,-115.736,-537.600,180.00,0.00,180.00
C00686=1566.309,-122.906,-537.600,180.00,-0.00,-180.00
C00687=1564.369,-129.889,-537.600,180.00,0.00,180.00
C00688=1561.677,-136.648,-537.600,180.00,0.00,-180.00
C00689=1558.273,-143.069,-537.600,180.00,-0.00,-180.00
C00690=1554.199,-149.078,-537.600,180.00,0.00,-180.00
C00691=1549.497,-154.613,-537.600,180.00,-0.00,-180.00
C00692=1544.220,-159.611,-537.600,180.00,-0.00,-180.00
C00693=1538.438,-164.005,-537.600,180.00,0.00,180.00
C00694=1532.217,-167.748,-537.600,180.00,-0.00,180.00
C00695=1525.621,-170.799,-537.600,180.00,-0.00,180.00
C00696=1518.745,-173.117,-537.600,180.00,0.00,180.00
C00697=1511.648,-174.680,-537.600,180.00,-0.00,180.00
C00698=1504.425,-175.465,-537.600,180.00,0.00,-180.00
C00699=1497.169,-175.466,-537.600,180.00,0.00,-180.00
C00700=1489.946,-174.680,-537.600,180.00,0.00,-180.00
C00701=1482.849,-173.117,-537.600,180.00,0.00,-180.00
C00702=1475.973,-170.799,-537.600,180.00,0.00,-180.00
C00703=1469.377,-167.748,-537.600,180.00,-0.00,180.00
C00704=1463.157,-164.006,-537.600,180.00,0.00,-180.00
C00705=1457.370,-159.607,-537.600,180.00,0.00,-180.00
C00706=1452.096,-154.612,-537.600,180.00,-0.00,-180.00
C00707=1447.394,-149.078,-537.600,180.00,0.00,-180.00
C00708=1443.319,-143.068,-537.600,180.00,0.00,-180.00
C00709=1439.916,-136.648,-537.600,180.00,0.00,-180.00
C00710=1437.217,-129.875,-537.600,180.00,-0.00,-180.00
C00711=1435.285,-122.905,-537.600,180.00,0.00,180.00
C00712=1434.110,-115.732,-537.600,180.00,-0.00,180.00
C00713=1433.717,-108.482,-537.600,180.00,-0.00,-180.00
C00714=1447.095,-146.858,-537.600,180.00,0.00,180.00
C00715=1462.456,-162.219,-537.600,180.00,0.00,-180.00
C00716=1462.809,-162.572,-537.600,180.00,0.00,180.00
C00717=1470.003,-166.937,-537.600,180.00,0.00,-180.00
C00718=1442.550,-139.485,-537.600,180.00,0.00,-180.00
C00719=1442.197,-139.132,-537.600,180.00,0.00,-180.00
C00720=1439.965,-134.071,-537.600,180.00,-0.00,-180.00
C00721=1475.264,-169.370,-537.600,180.00,-0.00,180.00
C00722=1475.617,-169.723,-537.600,180.00,0.00,180.00
C00723=1479.735,-171.013,-537.600,180.00,0.00,-180.00
C00724=1438.122,-129.400,-537.600,180.00,0.00,180.00
C00725=1437.769,-129.047,-537.600,180.00,0.00,180.00
C00726=1437.038,-125.487,-537.600,180.00,-0.00,-180.00
C00727=1483.869,-172.318,-537.600,180.00,-0.00,-180.00
C00728=1487.497,-173.117,-537.600,180.00,-0.00,-180.00
C00729=1436.105,-121.726,-537.600,180.00,0.00,180.00
C00730=1435.551,-118.344,-537.600,180.00,-0.00,180.00
C00731=1490.997,-173.789,-537.600,180.00,-0.00,-180.00
C00732=1494.171,-174.135,-537.600,180.00,0.00,-180.00
C00733=1435.074,-115.038,-537.600,180.00,-0.00,-180.00
C00734=1434.911,-112.047,-537.600,180.00,-0.00,180.00
C00735=1497.331,-174.467,-537.600,180.00,-0.00,-180.00
C00736=1500.160,-174.467,-537.600,180.00,0.00,180.00
C00737=1434.749,-109.056,-537.600,180.00,-0.00,-180.00
C00738=1434.836,-106.314,-537.600,180.00,0.00,180.00
C00739=1502.987,-174.466,-537.600,180.00,0.00,-180.00
C00740=1505.674,-174.324,-537.600,180.00,-0.00,-180.00
C00741=1434.981,-103.631,-537.600,180.00,-0.00,-180.00
C00742=1435.164,-100.986,-537.600,180.00,0.00,-180.00
C00743=1508.225,-174.047,-537.600,180.00,0.00,180.00
C00744=1510.776,-173.769,-537.600,180.00,0.00,-180.00
C00745=1435.563,-98.556,-537.600,180.00,0.00,-180.00
C00746=1435.961,-96.126,-537.600,180.00,-0.00,-180.00
C00747=1513.159,-173.324,-537.600,180.00,-0.00,-180.00
C00748=1515.477,-172.813,-537.600,180.00,0.00,-180.00
C00749=1436.411,-93.748,-537.600,180.00,0.00,-180.00
C00750=1437.026,-91.534,-537.600,180.00,0.00,-180.00
C00751=1517.795,-172.303,-537.600,180.00,-0.00,-180.00
C00752=1519.970,-171.649,-537.600,180.00,-0.00,180.00
C00753=1437.641,-89.320,-537.600,180.00,-0.00,-180.00
C00754=1438.281,-87.132,-537.600,180.00,0.00,-180.00
C00755=1522.085,-170.936,-537.600,180.00,-0.00,180.00
C00756=1524.200,-170.223,-537.600,180.00,0.00,-180.00
C00757=1439.086,-85.109,-537.600,180.00,-0.00,-180.00
C00758=1439.892,-83.086,-537.600,180.00,0.00,-180.00
C00759=1526.224,-169.419,-537.600,180.00,0.00,180.00
C00760=1528.158,-168.524,-537.600,180.00,0.00,-180.00
C00761=1440.698,-81.063,-537.600,180.00,-0.00,-180.00
C00762=1441.649,-79.187,-537.600,180.00,-0.00,-180.00
C00763=1530.092,-167.630,-537.600,180.00,0.00,-180.00
C00764=1532.001,-166.710,-537.600,180.00,0.00,180.00
C00765=1442.629,-77.338,-537.600,180.00,0.00,-180.00
C00766=1443.609,-75.489,-537.600,180.00,0.00,180.00
C00767=1533.768,-165.648,-537.600,180.00,0.00,-180.00
C00768=1535.533,-164.585,-537.600,180.00,-0.00,180.00
C00769=1444.657,-73.710,-537.600,180.00,0.00,-180.00
C00770=1445.800,-72.024,-537.600,180.00,-0.00,-180.00
C00771=1537.299,-163.523,-537.600,180.00,0.00,180.00
C00772=1538.959,-162.354,-537.600,180.00,0.00,180.00
C00773=1446.943,-70.338,-537.600,180.00,0.00,-180.00
C00774=1448.085,-68.652,-537.600,180.00,-0.00,-180.00
C00775=1540.566,-161.133,-537.600,180.00,0.00,-180.00
C00776=1542.173,-159.912,-537.600,180.00,-0.00,-180.00
C00777=1449.371,-67.109,-537.600,180.00,-0.00,-180.00
C00778=1450.671,-65.581,-537.600,180.00,0.00,180.00
C00779=1543.760,-158.671,-537.600,180.00,0.00,180.00
C00780=1545.212,-157.294,-537.600,180.00,-0.00,-180.00
C00781=1451.970,-64.051,-537.600,180.00,0.00,-180.00
C00782=1453.321,-62.574,-537.600,180.00,0.00,-180.00
C00783=1546.665,-155.918,-537.600,180.00,0.00,180.00
C00784=1548.117,-154.542,-537.600,180.00,-0.00,180.00
C00785=1454.773,-61.198,-537.600,180.00,0.00,-180.00
C00786=1456.226,-59.822,-537.600,180.00,-0.00,-180.00
C00787=1549.484,-153.081,-537.600,180.00,0.00,-180.00
C00788=1550.784,-151.552,-537.600,180.00,0.00,180.00
C00789=1457.678,-58.446,-537.600,180.00,-0.00,-180.00
C00790=1459.249,-57.189,-537.600,180.00,0.00,-180.00
C00791=1552.083,-150.023,-537.600,180.00,0.00,180.00
C00792=1553.383,-148.494,-537.600,180.00,-0.00,180.00
C00793=1460.856,-55.968,-537.600,180.00,-0.00,180.00
C00794=1462.463,-54.746,-537.600,180.00,0.00,-180.00
C00795=1554.528,-146.810,-537.600,180.00,-0.00,180.00
C00796=1555.670,-145.124,-537.600,180.00,0.00,-180.00
C00797=1464.105,-53.559,-537.600,180.00,0.00,-180.00
C00798=1465.871,-52.497,-537.600,180.00,-0.00,180.00
C00799=1556.813,-143.439,-537.600,180.00,0.00,-180.00
C00800=1557.879,-141.676,-537.600,180.00,0.00,180.00
C00801=1467.637,-51.434,-537.600,180.00,0.00,-180.00
C00802=1469.403,-50.372,-537.600,180.00,-0.00,-180.00
C00803=1558.859,-139.828,-537.600,180.00,0.00,-180.00
C00804=1559.838,-137.978,-537.600,180.00,0.00,-180.00
C00805=1471.295,-49.435,-537.600,180.00,0.00,180.00
C00806=1473.229,-48.541,-537.600,180.00,-0.00,180.00
C00807=1560.809,-136.121,-537.600,180.00,0.00,-180.00
C00808=1561.614,-134.098,-537.600,180.00,-0.00,-180.00
C00809=1475.163,-47.646,-537.600,180.00,0.00,-180.00
C00810=1477.167,-46.823,-537.600,180.00,0.00,-180.00
C00811=1562.420,-132.076,-537.600,180.00,0.00,-180.00
C00812=1563.226,-130.053,-537.600,180.00,0.00,180.00
C00813=1479.282,-46.109,-537.600,180.00,0.00,-180.00
C00814=1481.398,-45.396,-537.600,180.00,0.00,180.00
C00815=1563.886,-127.885,-537.600,180.00,0.00,-180.00
C00816=1564.501,-125.671,-537.600,180.00,-0.00,-180.00
C00817=1483.551,-44.721,-537.600,180.00,0.00,-180.00
C00818=1485.869,-44.210,-537.600,180.00,-0.00,-180.00
C00819=1565.117,-123.458,-537.600,180.00,-0.00,180.00
C00820=1565.590,-121.103,-537.600,180.00,0.00,180.00
C00821=1488.187,-43.700,-537.600,180.00,0.00,-180.00
C00822=1490.544,-43.229,-537.600,180.00,0.00,-180.00
C00823=1565.988,-118.672,-537.600,180.00,0.00,-180.00
C00824=1566.386,-116.242,-537.600,180.00,-0.00,-180.00
C00825=1493.095,-42.951,-537.600,180.00,0.00,-180.00
C00826=1495.645,-42.673,-537.600,180.00,-0.00,-180.00
C00827=1566.596,-113.624,-537.600,180.00,-0.00,-180.00
C00828=1566.741,-110.941,-537.600,180.00,0.00,180.00
C00829=1498.303,-42.502,-537.600,180.00,-0.00,180.00
C00830=1501.131,-42.502,-537.600,180.00,0.00,180.00
C00831=1566.861,-108.232,-537.600,180.00,0.00,-180.00
C00832=1566.698,-105.241,-537.600,180.00,0.00,-180.00
C00833=1503.960,-42.502,-537.600,180.00,-0.00,180.00
C00834=1507.083,-42.797,-537.600,180.00,0.00,-180.00
C00835=1566.536,-102.250,-537.600,180.00,0.00,-180.00
C00836=1566.100,-98.986,-537.600,180.00,-0.00,-180.00
C00837=1510.257,-43.143,-537.600,180.00,0.00,180.00
C00838=1513.709,-43.766,-537.600,180.00,0.00,180.00
C00839=1565.545,-95.602,-537.600,180.00,-0.00,-180.00
C00840=1564.668,-91.897,-537.600,180.00,0.00,-180.00
C00841=1517.337,-44.566,-537.600,180.00,-0.00,-180.00
C00842=1516.984,-44.213,-537.600,180.00,-0.00,180.00
C00843=1521.403,-45.804,-537.600,180.00,0.00,-180.00
C00844=1563.583,-87.984,-537.600,180.00,-0.00,-180.00
C00845=1563.936,-88.337,-537.600,180.00,-0.00,-180.00
C00846=1561.825,-83.397,-537.600,180.00,0.00,180.00
C00847=1525.768,-47.340,-537.600,180.00,0.00,-180.00
C00848=1525.415,-46.987,-537.600,180.00,-0.00,-180.00
C00849=1531.031,-49.775,-537.600,180.00,-0.00,-180.00
C00850=1559.380,-78.123,-537.600,180.00,-0.00,180.00
C00851=1559.733,-78.476,-537.600,180.00,-0.00,-180.00
C00852=1555.133,-71.048,-537.600,180.00,-0.00,-180.00
C00853=1537.886,-53.801,-537.600,180.00,0.00,180.00
C00854=1537.533,-53.448,-537.600,180.00,-0.00,-180.00
C00855=1537.533,-53.448,-536.400,180.00,0.00,-180.00
C00856=1440.075,-154.636,-536.400,180.00,-0.00,-180.00
C00857=1437.910,-156.296,-536.400,180.00,0.00,180.00
C00858=1443.440,-162.807,-536.400,180.00,0.00,-180.00
C00859=1449.657,-168.696,-536.400,180.00,0.00,-180.00
C00860=1456.460,-173.867,-536.400,180.00,-0.00,-180.00
C00861=1463.793,-178.279,-536.400,180.00,0.00,180.00
C00862=1471.559,-181.872,-536.400,180.00,0.00,180.00
C00863=1479.662,-184.602,-536.400,180.00,-0.00,180.00
C00864=1488.021,-186.442,-536.400,180.00,0.00,180.00
C00865=1496.519,-187.367,-536.400,180.00,-0.00,-180.00
C00866=1505.075,-187.367,-536.400,180.00,-0.00,-180.00
C00867=1513.573,-186.442,-536.400,180.00,-0.00,180.00
C00868=1521.932,-184.602,-536.400,180.00,0.00,-180.00
C00869=1530.035,-181.872,-536.400,180.00,-0.00,-180.00
C00870=1537.801,-178.279,-536.400,180.00,0.00,180.00
C00871=1545.134,-173.867,-536.400,180.00,-0.00,-180.00
C00872=1551.937,-168.696,-536.400,180.00,-0.00,-180.00
C00873=1558.154,-162.807,-536.400,180.00,0.00,180.00
C00874=1563.684,-156.296,-536.400,180.00,-0.00,180.00
C00875=1568.487,-149.212,-536.400,180.00,0.00,-180.00
C00876=1572.495,-141.652,-536.400,180.00,0.00,-180.00
C00877=1575.658,-133.713,-536.400,180.00,0.00,180.00
C00878=1577.949,-125.463,-536.400,180.00,0.00,180.00
C00879=1579.332,-117.028,-536.400,180.00,-0.00,180.00
C00880=1579.795,-108.484,-536.400,180.00,-0.00,-180.00
C00881=1579.332,-99.940,-536.400,180.00,0.00,-180.00
C00882=1577.949,-91.505,-536.400,180.00,0.00,-180.00
C00883=1575.658,-83.255,-536.400,180.00,-0.00,-180.00
C00884=1572.495,-75.316,-536.400,180.00,-0.00,-180.00
C00885=1568.487,-67.756,-536.400,180.00,0.00,180.00
C00886=1563.684,-60.672,-536.400,180.00,-0.00,-180.00
C00887=1558.154,-54.161,-536.400,180.00,-0.00,180.00
C00888=1551.937,-48.272,-536.400,180.00,-0.00,-180.00
C00889=1545.134,-43.101,-536.400,180.00,0.00,-180.00
C00890=1537.801,-38.689,-536.400,180.00,-0.00,-180.00
C00891=1530.035,-35.096,-536.400,180.00,-0.00,-180.00
C00892=1521.932,-32.366,-536.400,180.00,-0.00,180.00
C00893=1513.573,-30.526,-536.400,180.00,-0.00,-180.00
C00894=1505.075,-29.601,-536.400,180.00,0.00,-180.00
C00895=1496.519,-29.601,-536.400,180.00,0.00,-180.00
C00896=1488.021,-30.526,-536.400,180.00,0.00,-180.00
C00897=1479.662,-32.366,-536.400,180.00,0.00,-180.00
C00898=1471.559,-35.096,-536.400,180.00,-0.00,-180.00
C00899=1463.793,-38.689,-536.400,180.00,-0.00,-180.00
C00900=1456.460,-43.101,-536.400,180.00,-0.00,-180.00
C00901=1449.657,-48.272,-536.400,180.00,0.00,-180.00
C00902=1443.440,-54.161,-536.400,180.00,0.00,-180.00
C00903=1437.910,-60.672,-536.400,180.00,-0.00,-180.00
C00904=1433.107,-67.756,-536.400,180.00,0.00,-180.00
C00905=1429.099,-75.316,-536.400,180.00,0.00,-180.00
C00906=1425.936,-83.255,-536.400,180.00,0.00,180.00
C00907=1423.645,-91.505,-536.400,180.00,-0.00,180.00
C00908=1422.262,-99.940,-536.400,180.00,-0.00,-180.00
C00909=1421.799,-108.484,-536.400,180.00,0.00,-180.00
C00910=1422.262,-117.028,-536.400,180.00,-0.00,-180.00
C00911=1423.645,-125.463,-536.400,180.00,0.00,-180.00
C00912=1425.936,-133.713,-536.400,180.00,-0.00,-180.00
C00913=1429.099,-141.652,-536.400,180.00,0.00,-180.00
C00914=1433.107,-149.212,-536.400,180.00,0.00,-180.00
C00915=1437.910,-156.296,-536.400,180.00,0.00,180.00
C00916=1443.440,-162.807,-536.379,180.00,0.00,-180.00
C00917=1449.657,-168.696,-536.359,180.00,-0.00,-180.00
C00918=1456.460,-173.867,-536.338,180.00,0.00,-180.00
C00919=1463.793,-178.279,-536.317,180.00,0.00,180.00
C00920=1471.559,-181.872,-536.297,180.00,-0.00,180.00
C00921=1479.662,-184.602,-536.276,180.00,-0.00,180.00
C00922=1488.021,-186.442,-536.255,180.00,-0.00,180.00
C00923=1496.519,-187.367,-536.234,180.00,0.00,-180.00
C00924=1505.075,-187.367,-536.214,180.00,-0.00,-180.00
C00925=1513.573,-186.442,-536.193,180.00,-0.00,180.00
C00926=1521.932,-184.602,-536.172,180.00,0.00,-180.00
C00927=1530.035,-181.872,-536.152,180.00,-0.00,-180.00
C00928=1537.801,-178.279,-536.131,180.00,0.00,180.00
C00929=1545.134,-173.867,-536.110,180.00,0.00,-180.00
C00930=1551.937,-168.696,-536.090,180.00,0.00,-180.00
C00931=1558.154,-162.807,-536.069,180.00,-0.00,180.00
C00932=1563.684,-156.296,-536.048,180.00,-0.00,180.00
C00933=1568.487,-149.212,-536.028,180.00,0.00,-180.00
C00934=1572.495,-141.652,-536.007,180.00,0.00,-180.00
C00935=1575.658,-133.713,-535.986,180.00,-0.00,180.00
C00936=1577.949,-125.463,-535.966,180.00,0.00,180.00
C00937=1579.332,-117.028,-535.945,180.00,-0.00,180.00
C00938=1579.795,-108.484,-535.924,180.00,-0.00,-180.00
C00939=1579.332,-99.940,-535.903,180.00,0.00,-180.00
C00940=1577.949,-91.505,-535.883,180.00,-0.00,-180.00
C00941=1575.658,-83.255,-535.862,180.00,-0.00,-180.00
C00942=1572.495,-75.316,-535.841,180.00,0.00,-180.00
C00943=1568.487,-67.756,-535.821,180.00,0.00,180.00
C00944=1563.684,-60.672,-535.800,180.00,-0.00,-180.00
C00945=1558.154,-54.161,-535.779,180.00,0.00,180.00
C00946=1551.937,-48.272,-535.759,180.00,0.00,-180.00
C00947=1545.134,-43.101,-535.738,180.00,-0.00,-180.00
C00948=1537.801,-38.689,-535.717,180.00,-0.00,-180.00
C00949=1530.035,-35.096,-535.697,180.00,-0.00,-180.00
C00950=1521.932,-32.366,-535.676,180.00,0.00,180.00
C00951=1513.573,-30.526,-535.655,180.00,0.00,-180.00
C00952=1505.075,-29.601,-535.634,180.00,0.00,-180.00
C00953=1496.519,-29.601,-535.614,180.00,0.00,-180.00
C00954=1488.021,-30.526,-535.593,180.00,0.00,-180.00
C00955=1479.662,-32.366,-535.572,180.00,0.00,-180.00
C00956=1471.559,-35.096,-535.552,180.00,0.00,-180.00
C00957=1463.793,-38.689,-535.531,180.00,-0.00,-180.00
C00958=1456.460,-43.101,-535.510,180.00,0.00,-180.00
C00959=1449.657,-48.272,-535.490,180.00,0.00,-180.00
C00960=1443.440,-54.161,-535.469,180.00,0.00,-180.00
C00961=1437.910,-60.672,-535.448,180.00,-0.00,-180.00
C00962=1433.107,-67.756,-535.428,180.00,0.00,-180.00
C00963=1429.099,-75.316,-535.407,180.00,0.00,-180.00
C00964=1425.936,-83.255,-535.386,180.00,0.00,180.00
C00965=1423.645,-91.505,-535.366,180.00,0.00,180.00
C00966=1422.262,-99.940,-535.345,180.00,-0.00,-180.00
C00967=1421.799,-108.484,-535.324,180.00,0.00,-180.00
C00968=1422.262,-117.028,-535.303,180.00,0.00,-180.00
C00969=1423.645,-125.463,-535.283,180.00,-0.00,-180.00
C00970=1425.936,-133.713,-535.262,180.00,-0.00,-180.00
C00971=1429.099,-141.652,-535.241,180.00,0.00,-180.00
C00972=1433.107,-149.212,-535.221,180.00,0.00,-180.00
C00973=1437.910,-156.296,-535.200,180.00,-0.00,180.00
C00974=1443.440,-162.807,-535.179,180.00,0.00,-180.00
C00975=1449.657,-168.696,-535.159,180.00,0.00,-180.00
C00976=1456.460,-173.867,-535.138,180.00,0.00,-180.00
C00977=1463.793,-178.279,-535.117,180.00,-0.00,180.00
C00978=1471.559,-181.872,-535.097,180.00,0.00,180.00
C00979=1479.662,-184.602,-535.076,180.00,-0.00,180.00
C00980=1488.021,-186.442,-535.055,180.00,-0.00,180.00
C00981=1496.519,-187.367,-535.034,180.00,-0.00,-180.00
C00982=1505.075,-187.367,-535.014,180.00,-0.00,-180.00
C00983=1513.573,-186.442,-534.993,180.00,-0.00,180.00
C00984=1521.932,-184.602,-534.972,180.00,0.00,-180.00
C00985=1530.035,-181.872,-534.952,180.00,-0.00,-180.00
C00986=1537.801,-178.279,-534.931,180.00,0.00,180.00
C00987=1545.134,-173.867,-534.910,180.00,0.00,-180.00
C00988=1551.937,-168.696,-534.890,180.00,0.00,-180.00
C00989=1558.154,-162.807,-534.869,180.00,-0.00,180.00
C00990=1563.684,-156.296,-534.848,180.00,0.00,180.00
C00991=1568.487,-149.212,-534.828,180.00,-0.00,-180.00
C00992=1572.495,-141.652,-534.807,180.00,-0.00,-180.00
C00993=1575.658,-133.713,-534.786,180.00,0.00,180.00
C00994=1577.949,-125.463,-534.766,180.00,-0.00,180.00
C00995=1579.332,-117.028,-534.745,180.00,-0.00,180.00
C00996=1579.795,-108.484,-534.724,180.00,0.00,-180.00
C00997=1579.332,-99.940,-534.703,180.00,0.00,-180.00
C00998=1577.949,-91.505,-534.683,180.00,0.00,-180.00
C00999=1575.658,-83.255,-534.662,180.00,0.00,-180.00
C01000=1572.495,-75.316,-534.641,180.00,0.00,-180.00
C01001=1568.487,-67.756,-534.621,180.00,-0.00,180.00
C01002=1563.684,-60.672,-534.600,180.00,0.00,-180.00
C01003=1558.154,-54.161,-534.579,180.00,0.00,180.00
C01004=1551.937,-48.272,-534.559,180.00,-0.00,-180.00
C01005=1545.134,-43.101,-534.538,180.00,0.00,-180.00
C01006=1537.801,-38.689,-534.517,180.00,0.00,-180.00
C01007=1530.035,-35.096,-534.497,180.00,-0.00,-180.00
C01008=1521.932,-32.366,-534.476,180.00,0.00,180.00
C01009=1513.573,-30.526,-534.455,180.00,0.00,-180.00
C01010=1505.075,-29.601,-534.434,180.00,0.00,-180.00
C01011=1496.519,-29.601,-534.414,180.00,0.00,-180.00
C01012=1488.021,-30.526,-534.393,180.00,0.00,-180.00
C01013=1479.662,-32.366,-534.372,180.00,0.00,-180.00
C01014=1471.559,-35.096,-534.352,180.00,-0.00,-180.00
C01015=1463.793,-38.689,-534.331,180.00,-0.00,-180.00
C01016=1456.460,-43.101,-534.310,180.00,-0.00,-180.00
C01017=1449.657,-48.272,-534.290,180.00,-0.00,-180.00
C01018=1443.440,-54.161,-534.269,180.00,0.00,-180.00
C01019=1437.910,-60.672,-534.248,180.00,-0.00,-180.00
C01020=1433.107,-67.756,-534.228,180.00,-0.00,-180.00
C01021=1429.099,-75.316,-534.207,180.00,0.00,-180.00
C01022=1425.936,-83.255,-534.186,180.00,0.00,180.00
C01023=1423.645,-91.505,-534.166,180.00,0.00,180.00
C01024=1422.262,-99.940,-534.145,180.00,-0.00,-180.00
C01025=1421.799,-108.484,-534.124,180.00,0.00,-180.00
C01026=1422.262,-117.028,-534.103,180.00,-0.00,-180.00
C01027=1423.645,-125.463,-534.083,180.00,0.00,-180.00
C01028=1425.936,-133.713,-534.062,180.00,-0.00,-180.00
C01029=1429.099,-141.652,-534.041,180.00,0.00,-180.00
C01030=1433.107,-149.212,-534.021,180.00,0.00,-180.00
C01031=1437.910,-156.296,-534.000,180.00,0.00,180.00
C01032=1443.440,-162.807,-533.979,180.00,0.00,-180.00
C01033=1449.657,-168.696,-533.959,180.00,0.00,-180.00
C01034=1456.460,-173.867,-533.938,180.00,0.00,-180.00
C01035=1463.793,-178.279,-533.917,180.00,0.00,180.00
C01036=1471.559,-181.872,-533.897,180.00,0.00,180.00
C01037=1479.662,-184.602,-533.876,180.00,0.00,180.00
C01038=1488.021,-186.442,-533.855,180.00,0.00,180.00
C01039=1496.519,-187.367,-533.834,180.00,0.00,-180.00
C01040=1505.075,-187.367,-533.814,180.00,0.00,-180.00
C01041=1513.573,-186.442,-533.793,180.00,-0.00,180.00
C01042=1521.932,-184.602,-533.772,180.00,-0.00,-180.00
C01043=1530.035,-181.872,-533.752,180.00,-0.00,-180.00
C01044=1537.801,-178.279,-533.731,180.00,0.00,180.00
C01045=1545.134,-173.867,-533.710,180.00,-0.00,-180.00
C01046=1551.937,-168.696,-533.690,180.00,0.00,-180.00
C01047=1558.154,-162.807,-533.669,180.00,-0.00,180.00
C01048=1563.684,-156.296,-533.648,180.00,0.00,180.00
C01049=1568.487,-149.212,-533.628,180.00,0.00,-180.00
C01050=1572.495,-141.652,-533.607,180.00,0.00,-180.00
C01051=1575.658,-133.713,-533.586,180.00,0.00,180.00
C01052=1577.949,-125.463,-533.566,180.00,-0.00,180.00
C01053=1579.332,-117.028,-533.545,180.00,0.00,180.00
C01054=1579.795,-108.484,-533.524,180.00,0.00,-180.00
C01055=1579.332,-99.940,-533.503,180.00,-0.00,-180.00
C01056=1577.949,-91.505,-533.483,180.00,0.00,-180.00
C01057=1575.658,-83.255,-533.462,180.00,-0.00,-180.00
C01058=1572.495,-75.316,-533.441,180.00,0.00,-180.00
C01059=1568.487,-67.756,-533.421,180.00,0.00,180.00
C01060=1563.684,-60.672,-533.400,180.00,0.00,-180.00
C01061=1558.154,-54.161,-533.379,180.00,0.00,180.00
C01062=1551.937,-48.272,-533.359,180.00,0.00,-180.00
C01063=1545.134,-43.101,-533.338,180.00,0.00,-180.00
C01064=1537.801,-38.689,-533.317,180.00,0.00,-180.00
C01065=1530.035,-35.096,-533.297,180.00,0.00,-180.00
C01066=1521.932,-32.366,-533.276,180.00,-0.00,180.00
C01067=1513.573,-30.526,-533.255,180.00,-0.00,-180.00
C01068=1505.075,-29.601,-533.234,180.00,0.00,-180.00
C01069=1496.519,-29.601,-533.214,180.00,-0.00,-180.00
C01070=1488.021,-30.526,-533.193,180.00,0.00,-180.00
C01071=1479.662,-32.366,-533.172,180.00,0.00,-180.00
C01072=1471.559,-35.096,-533.152,180.00,0.00,-180.00
C01073=1463.793,-38.689,-533.131,180.00,-0.00,-180.00
C01074=1456.460,-43.101,-533.110,180.00,-0.00,-180.00
C01075=1449.657,-48.272,-533.090,180.00,0.00,-180.00
C01076=1443.440,-54.161,-533.069,180.00,0.00,-180.00
C01077=1437.910,-60.672,-533.048,180.00,-0.00,-180.00
C01078=1433.107,-67.756,-533.028,180.00,0.00,-180.00
C01079=1429.099,-75.316,-533.007,180.00,0.00,-180.00
C01080=1425.936,-83.255,-532.986,180.00,0.00,180.00
C01081=1423.645,-91.505,-532.966,180.00,-0.00,180.00
C01082=1422.262,-99.940,-532.945,180.00,-0.00,-180.00
C01083=1421.799,-108.484,-532.924,180.00,-0.00,-180.00
C01084=1422.262,-117.028,-532.903,180.00,-0.00,-180.00
C01085=1423.645,-125.463,-532.883,180.00,-0.00,-180.00
C01086=1425.936,-133.713,-532.862,180.00,0.00,-180.00
C01087=1429.099,-141.652,-532.841,180.00,-0.00,-180.00
C01088=1433.107,-149.212,-532.821,180.00,0.00,-180.00
C01089=1437.910,-156.296,-532.800,180.00,0.00,180.00
C01090=1443.440,-162.807,-532.779,180.00,-0.00,-180.00
C01091=1449.657,-168.696,-532.759,180.00,-0.00,-180.00
C01092=1456.460,-173.867,-532.738,180.00,-0.00,-180.00
C01093=1463.793,-178.279,-532.717,180.00,0.00,180.00
C01094=1471.559,-181.872,-532.697,180.00,0.00,180.00
C01095=1479.662,-184.602,-532.676,180.00,0.00,180.00
C01096=1488.021,-186.442,-532.655,180.00,-0.00,180.00
C01097=1496.519,-187.367,-532.634,180.00,0.00,-180.00
C01098=1505.075,-187.367,-532.614,180.00,-0.00,-180.00
C01099=1513.573,-186.442,-532.593,180.00,-0.00,180.00
C01100=1521.932,-184.602,-532.572,180.00,0.00,-180.00
C01101=1530.035,-181.872,-532.552,180.00,0.00,-180.00
C01102=1537.801,-178.279,-532.531,180.00,-0.00,180.00
C01103=1545.134,-173.867,-532.510,180.00,-0.00,-180.00
C01104=1551.937,-168.696,-532.490,180.00,-0.00,-180.00
C01105=1558.154,-162.807,-532.469,180.00,0.00,180.00
C01106=1563.684,-156.296,-532.448,180.00,-0.00,180.00
C01107=1568.487,-149.212,-532.428,180.00,-0.00,-180.00
C01108=1572.495,-141.652,-532.407,180.00,0.00,-180.00
C01109=1575.658,-133.713,-532.386,180.00,0.00,180.00
C01110=1577.949,-125.463,-532.366,180.00,-0.00,180.00
C01111=1579.332,-117.028,-532.345,180.00,-0.00,180.00
C01112=1579.795,-108.484,-532.324,180.00,-0.00,-180.00
C01113=1579.332,-99.940,-532.303,180.00,0.00,-180.00
C01114=1577.949,-91.505,-532.283,180.00,0.00,-180.00
C01115=1575.658,-83.255,-532.262,180.00,-0.00,-180.00
C01116=1572.495,-75.316,-532.241,180.00,0.00,-180.00
C01117=1568.487,-67.756,-532.221,180.00,-0.00,180.00
C01118=1563.684,-60.672,-532.200,180.00,0.00,-180.00
C01119=1558.154,-54.161,-532.179,180.00,0.00,180.00
C01120=1551.937,-48.272,-532.159,180.00,-0.00,-180.00
C01121=1545.134,-43.101,-532.138,180.00,-0.00,-180.00
C01122=1537.801,-38.689,-532.117,180.00,-0.00,-180.00
C01123=1530.035,-35.096,-532.097,180.00,-0.00,-180.00
C01124=1521.932,-32.366,-532.076,180.00,0.00,180.00
C01125=1513.573,-30.526,-532.055,180.00,0.00,-180.00
C01126=1505.075,-29.601,-532.034,180.00,0.00,-180.00
C01127=1496.519,-29.601,-532.014,180.00,-0.00,-180.00
C01128=1488.021,-30.526,-531.993,180.00,0.00,-180.00
C01129=1479.662,-32.366,-531.972,180.00,-0.00,-180.00
C01130=1471.559,-35.096,-531.952,180.00,-0.00,-180.00
C01131=1463.793,-38.689,-531.931,180.00,-0.00,-180.00
C01132=1456.460,-43.101,-531.910,180.00,-0.00,-180.00
C01133=1449.657,-48.272,-531.890,180.00,0.00,-180.00
C01134=1443.440,-54.161,-531.869,180.00,0.00,-180.00
C01135=1437.910,-60.672,-531.848,180.00,0.00,-180.00
C01136=1433.107,-67.756,-531.828,180.00,-0.00,-180.00
C01137=1429.099,-75.316,-531.807,180.00,0.00,-180.00
C01138=1425.936,-83.255,-531.786,180.00,0.00,180.00
C01139=1423.645,-91.505,-531.766,180.00,0.00,180.00
C01140=1422.262,-99.940,-531.745,180.00,-0.00,-180.00
C01141=1421.799,-108.484,-531.724,180.00,-0.00,-180.00
C01142=1422.262,-117.028,-531.703,180.00,-0.00,-180.00
C01143=1423.645,-125.463,-531.683,180.00,-0.00,-180.00
C01144=1425.936,-133.713,-531.662,180.00,-0.00,-180.00
C01145=1429.099,-141.652,-531.641,180.00,0.00,-180.00
C01146=1433.107,-149.212,-531.621,180.00,0.00,-180.00
C01147=1437.910,-156.296,-531.600,180.00,0.00,180.00
C01148=1443.440,-162.807,-531.579,180.00,0.00,-180.00
C01149=1449.657,-168.696,-531.559,180.00,0.00,-180.00
C01150=1456.460,-173.867,-531.538,180.00,-0.00,-180.00
C01151=1463.793,-178.279,-531.517,180.00,0.00,180.00
C01152=1471.559,-181.872,-531.497,180.00,-0.00,180.00
C01153=1479.662,-184.602,-531.476,180.00,0.00,180.00
C01154=1488.021,-186.442,-531.455,180.00,-0.00,180.00
C01155=1496.519,-187.367,-531.434,180.00,0.00,-180.00
C01156=1505.075,-187.367,-531.414,180.00,0.00,-180.00
C01157=1513.573,-186.442,-531.393,180.00,0.00,180.00
C01158=1521.932,-184.602,-531.372,180.00,0.00,-180.00
C01159=1530.035,-181.872,-531.352,180.00,0.00,-180.00
C01160=1537.801,-178.279,-531.331,180.00,0.00,180.00
C01161=1545.134,-173.867,-531.310,180.00,0.00,-180.00
C01162=1551.937,-168.696,-531.290,180.00,0.00,-180.00
C01163=1558.154,-162.807,-531.269,180.00,0.00,180.00
C01164=1563.684,-156.296,-531.248,180.00,0.00,180.00
C01165=1568.487,-149.212,-531.228,180.00,0.00,-180.00
C01166=1572.495,-141.652,-531.207,180.00,0.00,-180.00
C01167=1575.658,-133.713,-531.186,180.00,0.00,180.00
C01168=1577.949,-125.463,-531.166,180.00,0.00,180.00
C01169=1579.332,-117.028,-531.145,180.00,0.00,180.00
C01170=1579.795,-108.484,-531.124,180.00,-0.00,-180.00
C01171=1579.332,-99.940,-531.103,180.00,0.00,-180.00
C01172=1577.949,-91.505,-531.083,180.00,-0.00,-180.00
C01173=1575.658,-83.255,-531.062,180.00,-0.00,-180.00
C01174=1572.495,-75.316,-531.041,180.00,0.00,-180.00
C01175=1568.487,-67.756,-531.021,180.00,0.00,180.00
C01176=1563.684,-60.672,-531.000,180.00,0.00,-180.00
C01177=1558.154,-54.161,-530.979,180.00,-0.00,180.00
C01178=1551.937,-48.272,-530.959,180.00,-0.00,-180.00
C01179=1545.134,-43.101,-530.938,180.00,0.00,-180.00
C01180=1537.801,-38.689,-530.917,180.00,-0.00,-180.00
C01181=1530.035,-35.096,-530.897,180.00,0.00,-180.00
C01182=1521.932,-32.366,-530.876,180.00,-0.00,180.00
C01183=1513.573,-30.526,-530.855,180.00,0.00,-180.00
C01184=1505.075,-29.601,-530.834,180.00,0.00,-180.00
C01185=1496.519,-29.601,-530.814,180.00,0.00,-180.00
C01186=1488.021,-30.526,-530.793,180.00,0.00,-180.00
C01187=1479.662,-32.366,-530.772,180.00,0.00,-180.00
C01188=1471.559,-35.096,-530.752,180.00,0.00,-180.00
C01189=1463.793,-38.689,-530.731,180.00,-0.00,-180.00
C01190=1456.460,-43.101,-530.710,180.00,-0.00,-180.00
C01191=1449.657,-48.272,-530.690,180.00,0.00,-180.00
C01192=1443.440,-54.161,-530.669,180.00,0.00,-180.00
C01193=1437.910,-60.672,-530.648,180.00,-0.00,-180.00
C01194=1433.107,-67.756,-530.628,180.00,-0.00,-180.00
C01195=1429.099,-75.316,-530.607,180.00,-0.00,-180.00
C01196=1425.936,-83.255,-530.586,180.00,-0.00,180.00
C01197=1423.645,-91.505,-530.566,180.00,0.00,180.00
C01198=1422.262,-99.940,-530.545,180.00,0.00,-180.00
C01199=1421.799,-108.484,-530.524,180.00,0.00,-180.00
C01200=1422.262,-117.028,-530.503,180.00,0.00,-180.00
C01201=1423.645,-125.463,-530.483,180.00,0.00,-180.00
C01202=1425.936,-133.713,-530.462,180.00,0.00,-180.00
C01203=1429.099,-141.652,-530.441,180.00,0.00,-180.00
C01204=1433.107,-149.212,-530.421,180.00,0.00,-180.00
C01205=1437.910,-156.296,-530.400,180.00,0.00,180.00
C01206=1443.440,-162.807,-530.379,180.00,0.00,-180.00
C01207=1449.657,-168.696,-530.359,180.00,-0.00,-180.00
C01208=1456.460,-173.867,-530.338,180.00,0.00,-180.00
C01209=1463.793,-178.279,-530.317,180.00,-0.00,180.00
C01210=1471.559,-181.872,-530.297,180.00,0.00,180.00
C01211=1479.662,-184.602,-530.276,180.00,0.00,180.00
C01212=1488.021,-186.442,-530.255,180.00,0.00,180.00
C01213=1496.519,-187.367,-530.234,180.00,-0.00,-180.00
C01214=1505.075,-187.367,-530.214,180.00,-0.00,180.00
C01215=1513.573,-186.442,-530.193,180.00,-0.00,180.00
C01216=1521.932,-184.602,-530.172,180.00,-0.00,-180.00
C01217=1530.035,-181.872,-530.152,180.00,0.00,-180.00
C01218=1537.801,-178.279,-530.131,180.00,-0.00,180.00
C01219=1545.134,-173.867,-530.110,180.00,0.00,-180.00
C01220=1551.937,-168.696,-530.090,180.00,0.00,-180.00
C01221=1558.154,-162.807,-530.069,180.00,-0.00,180.00
C01222=1563.684,-156.296,-530.048,180.00,0.00,180.00
C01223=1568.487,-149.212,-530.028,180.00,-0.00,-180.00
C01224=1572.495,-141.652,-530.007,180.00,-0.00,-180.00
C01225=1575.658,-133.713,-529.986,180.00,-0.00,180.00
C01226=1577.949,-125.463,-529.966,180.00,0.00,180.00
C01227=1579.332,-117.028,-529.945,180.00,0.00,180.00
C01228=1579.795,-108.484,-529.924,180.00,0.00,-180.00
C01229=1579.332,-99.940,-529.903,180.00,-0.00,-180.00
C01230=1577.949,-91.505,-529.883,180.00,-0.00,-180.00
C01231=1575.658,-83.255,-529.862,180.00,-0.00,-180.00
C01232=1572.495,-75.316,-529.841,180.00,0.00,-180.00
C01233=1568.487,-67.756,-529.821,180.00,0.00,180.00
C01234=1563.684,-60.672,-529.800,180.00,-0.00,-180.00
C01235=1558.154,-54.161,-529.779,180.00,0.00,180.00
C01236=1551.937,-48.272,-529.759,180.00,-0.00,-180.00
C01237=1545.134,-43.101,-529.738,180.00,-0.00,-180.00
C01238=1537.801,-38.689,-529.717,180.00,0.00,-180.00
C01239=1530.035,-35.096,-529.697,180.00,-0.00,-180.00
C01240=1521.932,-32.366,-529.676,180.00,-0.00,180.00
C01241=1513.573,-30.526,-529.655,180.00,-0.00,-180.00
C01242=1505.075,-29.601,-529.634,180.00,-0.00,-180.00
C01243=1496.519,-29.601,-529.614,180.00,0.00,-180.00
C01244=1488.021,-30.526,-529.593,180.00,0.00,-180.00
C01245=1479.662,-32.366,-529.572,180.00,0.00,-180.00
C01246=1471.559,-35.096,-529.552,180.00,-0.00,-180.00
C01247=1463.793,-38.689,-529.531,180.00,-0.00,-180.00
C01248=1456.460,-43.101,-529.510,180.00,0.00,-180.00
C01249=1449.657,-48.272,-529.490,180.00,0.00,-180.00
C01250=1443.440,-54.161,-529.469,180.00,0.00,-180.00
C01251=1437.910,-60.672,-529.448,180.00,0.00,-180.00
C01252=1433.107,-67.756,-529.428,180.00,0.00,-180.00
C01253=1429.099,-75.316,-529.407,180.00,0.00,-180.00
C01254=1425.936,-83.255,-529.386,180.00,-0.00,180.00
C01255=1423.645,-91.505,-529.366,180.00,-0.00,180.00
C01256=1422.262,-99.940,-529.345,180.00,-0.00,-180.00
C01257=1421.799,-108.484,-529.324,180.00,0.00,-180.00
C01258=1422.262,-117.028,-529.303,180.00,-0.00,-180.00
C01259=1423.645,-125.463,-529.283,180.00,0.00,-180.00
C01260=1425.936,-133.713,-529.262,180.00,0.00,-180.00
C01261=1429.099,-141.652,-529.241,180.00,-0.00,-180.00
C01262=1433.107,-149.212,-529.221,180.00,-0.00,-180.00
C01263=1437.910,-156.296,-529.200,180.00,0.00,180.00
C01264=1443.440,-162.807,-529.179,180.00,0.00,-180.00
C01265=1449.657,-168.696,-529.159,180.00,0.00,-180.00
C01266=1456.460,-173.867,-529.138,180.00,0.00,-180.00
C01267=1463.793,-178.279,-529.117,180.00,-0.00,180.00
C01268=1471.559,-181.872,-529.097,180.00,-0.00,180.00
C01269=1479.662,-184.602,-529.076,180.00,0.00,180.00
C01270=1488.021,-186.442,-529.055,180.00,0.00,180.00
C01271=1496.519,-187.367,-529.034,180.00,0.00,-180.00
C01272=1505.075,-187.367,-529.014,180.00,-0.00,-180.00
C01273=1513.573,-186.442,-528.993,180.00,0.00,180.00
C01274=1521.932,-184.602,-528.972,180.00,0.00,-180.00
C01275=1530.035,-181.872,-528.952,180.00,0.00,-180.00
C01276=1537.801,-178.279,-528.931,180.00,0.00,180.00
C01277=1545.134,-173.867,-528.910,180.00,0.00,-180.00
C01278=1551.937,-168.696,-528.890,180.00,0.00,-180.00
C01279=1558.154,-162.807,-528.869,180.00,-0.00,180.00
C01280=1563.684,-156.296,-528.848,180.00,-0.00,180.00
C01281=1568.487,-149.212,-528.828,180.00,0.00,-180.00
C01282=1572.495,-141.652,-528.807,180.00,0.00,-180.00
C01283=1575.658,-133.713,-528.786,180.00,0.00,180.00
C01284=1577.949,-125.463,-528.766,180.00,-0.00,180.00
C01285=1579.332,-117.028,-528.745,180.00,0.00,180.00
C01286=1579.795,-108.484,-528.724,180.00,-0.00,-180.00
C01287=1579.332,-99.940,-528.703,180.00,-0.00,-180.00
C01288=1577.949,-91.505,-528.683,180.00,-0.00,-180.00
C01289=1575.658,-83.255,-528.662,180.00,0.00,-180.00
C01290=1572.495,-75.316,-528.641,180.00,0.00,-180.00
C01291=1568.487,-67.756,-528.621,180.00,0.00,180.00
C01292=1563.684,-60.672,-528.600,180.00,0.00,-180.00
C01293=1558.154,-54.161,-528.579,180.00,0.00,180.00
C01294=1551.937,-48.272,-528.559,180.00,0.00,-180.00
C01295=1545.134,-43.101,-528.538,180.00,0.00,-180.00
C01296=1537.801,-38.689,-528.517,180.00,-0.00,-180.00
C01297=1530.035,-35.096,-528.497,180.00,0.00,-180.00
C01298=1521.932,-32.366,-528.476,180.00,0.00,180.00
C01299=1513.573,-30.526,-528.455,180.00,0.00,-180.00
C01300=1505.075,-29.601,-528.434,180.00,0.00,-180.00
C01301=1496.519,-29.601,-528.414,180.00,-0.00,-180.00
C01302=1488.021,-30.526,-528.393,180.00,-0.00,-180.00
C01303=1479.662,-32.366,-528.372,180.00,-0.00,-180.00
C01304=1471.559,-35.096,-528.352,180.00,-0.00,-180.00
C01305=1463.793,-38.689,-528.331,180.00,0.00,-180.00
C01306=1456.460,-43.101,-528.310,180.00,0.00,-180.00
C01307=1449.657,-48.272,-528.290,180.00,-0.00,-180.00
C01308=1443.440,-54.161,-528.269,180.00,0.00,-180.00
C01309=1437.910,-60.672,-528.248,180.00,0.00,-180.00
C01310=1433.107,-67.756,-528.228,180.00,-0.00,-180.00
C01311=1429.099,-75.316,-528.207,180.00,-0.00,-180.00
C01312=1425.936,-83.255,-528.186,180.00,0.00,180.00
C01313=1423.645,-91.505,-528.166,180.00,0.00,180.00
C01314=1422.262,-99.940,-528.145,180.00,0.00,-180.00
C01315=1421.799,-108.484,-528.124,180.00,-0.00,-180.00
C01316=1422.262,-117.028,-528.103,180.00,-0.00,-180.00
C01317=1423.645,-125.463,-528.083,180.00,0.00,-180.00
C01318=1425.936,-133.713,-528.062,180.00,-0.00,-180.00
C01319=1429.099,-141.652,-528.041,180.00,-0.00,-180.00
C01320=1433.107,-149.212,-528.021,180.00,0.00,-180.00
C01321=1437.910,-156.296,-528.000,180.00,-0.00,180.00
C01322=1443.440,-162.807,-527.979,180.00,-0.00,-180.00
C01323=1449.657,-168.696,-527.959,180.00,-0.00,-180.00
C01324=1456.460,-173.867,-527.938,180.00,0.00,-180.00
C01325=1463.793,-178.279,-527.917,180.00,-0.00,180.00
C01326=1471.559,-181.872,-527.897,180.00,0.00,180.00
C01327=1479.662,-184.602,-527.876,180.00,-0.00,180.00
C01328=1488.021,-186.442,-527.855,180.00,0.00,180.00
C01329=1496.519,-187.367,-527.834,180.00,-0.00,-180.00
C01330=1505.075,-187.367,-527.814,180.00,-0.00,-180.00
C01331=1513.573,-186.442,-527.793,180.00,0.00,180.00
C01332=1521.932,-184.602,-527.772,180.00,0.00,-180.00
C01333=1530.035,-181.872,-527.752,180.00,-0.00,-180.00
C01334=1537.801,-178.279,-527.731,180.00,0.00,-180.00
C01335=1545.134,-173.867,-527.710,180.00,0.00,-180.00
C01336=1551.937,-168.696,-527.690,180.00,0.00,-180.00
C01337=1558.154,-162.807,-527.669,180.00,0.00,180.00
C01338=1563.684,-156.296,-527.648,180.00,-0.00,180.00
C01339=1568.487,-149.212,-527.628,180.00,0.00,-180.00
C01340=1572.495,-141.652,-527.607,180.00,0.00,-180.00
C01341=1575.658,-133.713,-527.586,180.00,0.00,180.00
C01342=1577.949,-125.463,-527.566,180.00,-0.00,180.00
C01343=1579.332,-117.028,-527.545,180.00,-0.00,180.00
C01344=1579.795,-108.484,-527.524,180.00,0.00,-180.00
C01345=1579.332,-99.940,-527.503,180.00,-0.00,-180.00
C01346=1577.949,-91.505,-527.483,180.00,0.00,-180.00
C01347=1575.658,-83.255,-527.462,180.00,0.00,-180.00
C01348=1572.495,-75.316,-527.441,180.00,-0.00,-180.00
C01349=1568.487,-67.756,-527.421,180.00,0.00,180.00
C01350=1563.684,-60.672,-527.400,180.00,-0.00,-180.00
C01351=1558.154,-54.161,-527.379,180.00,-0.00,180.00
C01352=1551.937,-48.272,-527.359,180.00,-0.00,-180.00
C01353=1545.134,-43.101,-527.338,180.00,0.00,-180.00
C01354=1537.801,-38.689,-527.317,180.00,0.00,-180.00
C01355=1530.035,-35.096,-527.297,180.00,0.00,-180.00
C01356=1521.932,-32.366,-527.276,180.00,0.00,180.00
C01357=1513.573,-30.526,-527.255,180.00,0.00,-180.00
C01358=1505.075,-29.601,-527.234,180.00,0.00,-180.00
C01359=1496.519,-29.601,-527.214,180.00,0.00,-180.00
C01360=1488.021,-30.526,-527.193,180.00,-0.00,-180.00
C01361=1479.662,-32.366,-527.172,180.00,-0.00,-180.00
C01362=1471.559,-35.096,-527.152,180.00,0.00,-180.00
C01363=1463.793,-38.689,-527.131,180.00,0.00,-180.00
C01364=1456.460,-43.101,-527.110,180.00,-0.00,-180.00
C01365=1449.657,-48.272,-527.090,180.00,0.00,-180.00
C01366=1443.440,-54.161,-527.069,180.00,-0.00,-180.00
C01367=1437.910,-60.672,-527.048,180.00,0.00,-180.00
C01368=1433.107,-67.756,-527.028,180.00,-0.00,-180.00
C01369=1429.099,-75.316,-527.007,180.00,-0.00,-180.00
C01370=1425.936,-83.255,-526.986,180.00,0.00,180.00
C01371=1423.645,-91.505,-526.966,180.00,0.00,180.00
C01372=1422.262,-99.940,-526.945,180.00,0.00,-180.00
C01373=1421.799,-108.484,-526.924,180.00,0.00,-180.00
C01374=1422.262,-117.028,-526.903,180.00,0.00,-180.00
C01375=1423.645,-125.463,-526.883,180.00,0.00,-180.00
C01376=1425.936,-133.713,-526.862,180.00,0.00,-180.00
C01377=1429.099,-141.652,-526.841,180.00,0.00,-180.00
C01378=1433.107,-149.212,-526.821,180.00,0.00,-180.00
C01379=1437.910,-156.296,-526.800,180.00,0.00,180.00
C01380=1443.440,-162.807,-526.779,180.00,-0.00,-180.00
C01381=1449.657,-168.696,-526.759,180.00,0.00,-180.00
C01382=1456.460,-173.867,-526.738,180.00,-0.00,-180.00
C01383=1463.793,-178.279,-526.717,180.00,0.00,180.00
C01384=1471.559,-181.872,-526.697,180.00,-0.00,180.00
C01385=1479.662,-184.602,-526.676,180.00,0.00,180.00
C01386=1488.021,-186.442,-526.655,180.00,0.00,180.00
C01387=1496.519,-187.367,-526.634,180.00,0.00,-180.00
C01388=1505.075,-187.367,-526.614,180.00,-0.00,-180.00
C01389=1513.573,-186.442,-526.593,180.00,-0.00,180.00
C01390=1521.932,-184.602,-526.572,180.00,0.00,-180.00
C01391=1530.035,-181.872,-526.552,180.00,-0.00,-180.00
C01392=1537.801,-178.279,-526.531,180.00,0.00,180.00
C01393=1545.134,-173.867,-526.510,180.00,-0.00,-180.00
C01394=1551.937,-168.696,-526.490,180.00,-0.00,-180.00
C01395=1558.154,-162.807,-526.469,180.00,0.00,180.00
C01396=1563.684,-156.296,-526.448,180.00,-0.00,180.00
C01397=1568.487,-149.212,-526.428,180.00,-0.00,-180.00
C01398=1572.495,-141.652,-526.407,180.00,0.00,-180.00
C01399=1575.658,-133.713,-526.386,180.00,-0.00,180.00
C01400=1577.949,-125.463,-526.366,180.00,0.00,180.00
C01401=1579.332,-117.028,-526.345,180.00,0.00,180.00
C01402=1579.795,-108.484,-526.324,180.00,0.00,-180.00
C01403=1579.332,-99.940,-526.303,180.00,-0.00,-180.00
C01404=1577.949,-91.505,-526.283,180.00,0.00,-180.00
C01405=1575.658,-83.255,-526.262,180.00,-0.00,-180.00
C01406=1572.495,-75.316,-526.241,180.00,0.00,-180.00
C01407=1568.487,-67.756,-526.221,180.00,-0.00,180.00
C01408=1563.684,-60.672,-526.200,180.00,0.00,-180.00
C01409=1558.154,-54.161,-526.179,180.00,0.00,180.00
C01410=1551.937,-48.272,-526.159,180.00,-0.00,-180.00
C01411=1545.134,-43.101,-526.138,180.00,-0.00,-180.00
C01412=1537.801,-38.689,-526.117,180.00,-0.00,-180.00
C01413=1530.035,-35.096,-526.097,180.00,0.00,-180.00
C01414=1521.932,-32.366,-526.076,180.00,-0.00,180.00
C01415=1513.573,-30.526,-526.055,180.00,-0.00,-180.00
C01416=1505.075,-29.601,-526.034,180.00,-0.00,-180.00
C01417=1496.519,-29.601,-526.014,180.00,0.00,-180.00
C01418=1488.021,-30.526,-525.993,180.00,0.00,-180.00
C01419=1479.662,-32.366,-525.972,180.00,-0.00,-180.00
C01420=1471.559,-35.096,-525.952,180.00,-0.00,-180.00
C01421=1463.793,-38.689,-525.931,180.00,0.00,-180.00
C01422=1456.460,-43.101,-525.910,180.00,0.00,-180.00
C01423=1449.657,-48.272,-525.890,180.00,0.00,-180.00
C01424=1443.440,-54.161,-525.869,180.00,-0.00,-180.00
C01425=1437.910,-60.672,-525.848,180.00,-0.00,-180.00
C01426=1433.107,-67.756,-525.828,180.00,-0.00,-180.00
C01427=1429.099,-75.316,-525.807,180.00,0.00,-180.00
C01428=1425.936,-83.255,-525.786,180.00,0.00,180.00
C01429=1423.645,-91.505,-525.766,180.00,0.00,180.00
C01430=1422.262,-99.940,-525.745,180.00,-0.00,-180.00
C01431=1421.799,-108.484,-525.724,180.00,0.00,-180.00
C01432=1422.262,-117.028,-525.703,180.00,0.00,-180.00
C01433=1423.645,-125.463,-525.683,180.00,0.00,-180.00
C01434=1425.936,-133.713,-525.662,180.00,0.00,-180.00
C01435=1429.099,-141.652,-525.641,180.00,0.00,-180.00
C01436=1433.107,-149.212,-525.621,180.00,0.00,-180.00
C01437=1437.910,-156.296,-525.600,180.00,0.00,180.00
C01438=1443.440,-162.807,-525.579,180.00,-0.00,-180.00
C01439=1449.657,-168.696,-525.559,180.00,-0.00,-180.00
C01440=1456.460,-173.867,-525.538,180.00,-0.00,-180.00
C01441=1463.793,-178.279,-525.517,180.00,-0.00,180.00
C01442=1471.559,-181.872,-525.497,180.00,0.00,180.00
C01443=1479.662,-184.602,-525.476,180.00,0.00,180.00
C01444=1488.021,-186.442,-525.455,180.00,0.00,180.00
C01445=1496.519,-187.367,-525.434,180.00,0.00,-180.00
C01446=1505.075,-187.367,-525.414,180.00,0.00,-180.00
C01447=1513.573,-186.442,-525.393,180.00,0.00,180.00
C01448=1521.932,-184.602,-525.372,180.00,0.00,-180.00
C01449=1530.035,-181.872,-525.352,180.00,0.00,-180.00
C01450=1537.801,-178.279,-525.331,180.00,-0.00,180.00
C01451=1545.134,-173.867,-525.310,180.00,-0.00,-180.00
C01452=1551.937,-168.696,-525.290,180.00,0.00,-180.00
C01453=1558.154,-162.807,-525.269,180.00,-0.00,180.00
C01454=1563.684,-156.296,-525.248,180.00,-0.00,180.00
C01455=1568.487,-149.212,-525.228,180.00,0.00,-180.00
C01456=1572.495,-141.652,-525.207,180.00,0.00,-180.00
C01457=1575.658,-133.713,-525.186,180.00,0.00,180.00
C01458=1577.949,-125.463,-525.166,180.00,-0.00,180.00
C01459=1579.332,-117.028,-525.145,180.00,0.00,180.00
C01460=1579.795,-108.484,-525.124,180.00,0.00,-180.00
C01461=1579.332,-99.940,-525.103,180.00,0.00,-180.00
C01462=1577.949,-91.505,-525.083,180.00,0.00,-180.00
C01463=1575.658,-83.255,-525.062,180.00,0.00,-180.00
C01464=1572.495,-75.316,-525.041,180.00,0.00,-180.00
C01465=1568.487,-67.756,-525.021,180.00,0.00,180.00
C01466=1563.684,-60.672,-525.000,180.00,-0.00,-180.00
C01467=1558.154,-54.161,-524.979,180.00,0.00,180.00
C01468=1551.937,-48.272,-524.959,180.00,0.00,-180.00
C01469=1545.134,-43.101,-524.938,180.00,0.00,-180.00
C01470=1537.801,-38.689,-524.917,180.00,0.00,-180.00
C01471=1530.035,-35.096,-524.897,180.00,-0.00,-180.00
C01472=1521.932,-32.366,-524.876,180.00,0.00,180.00
C01473=1513.573,-30.526,-524.855,180.00,0.00,-180.00
C01474=1505.075,-29.601,-524.834,180.00,0.00,-180.00
C01475=1496.519,-29.601,-524.814,180.00,0.00,-180.00
C01476=1488.021,-30.526,-524.793,180.00,-0.00,-180.00
C01477=1479.662,-32.366,-524.772,180.00,-0.00,-180.00
C01478=1471.559,-35.096,-524.752,180.00,0.00,-180.00
C01479=1463.793,-38.689,-524.731,180.00,0.00,-180.00
C01480=1456.460,-43.101,-524.710,180.00,0.00,-180.00
C01481=1449.657,-48.272,-524.690,180.00,0.00,-180.00
C01482=1443.440,-54.161,-524.669,180.00,-0.00,-180.00
C01483=1437.910,-60.672,-524.648,180.00,0.00,-180.00
C01484=1433.107,-67.756,-524.628,180.00,0.00,-180.00
C01485=1429.099,-75.316,-524.607,180.00,0.00,-180.00
C01486=1425.936,-83.255,-524.586,180.00,-0.00,180.00
C01487=1423.645,-91.505,-524.566,180.00,0.00,180.00
C01488=1422.262,-99.940,-524.545,180.00,0.00,-180.00
C01489=1421.799,-108.484,-524.524,180.00,-0.00,-180.00
C01490=1422.262,-117.028,-524.503,180.00,0.00,-180.00
C01491=1423.645,-125.463,-524.483,180.00,-0.00,-180.00
C01492=1425.936,-133.713,-524.462,180.00,0.00,-180.00
C01493=1429.099,-141.652,-524.441,180.00,0.00,-180.00
C01494=1433.107,-149.212,-524.421,180.00,0.00,-180.00
C01495=1437.910,-156.296,-524.400,180.00,-0.00,180.00
C01496=1443.440,-162.807,-524.379,180.00,-0.00,-180.00
C01497=1449.657,-168.696,-524.359,180.00,-0.00,-180.00
C01498=1456.460,-173.867,-524.338,180.00,0.00,-180.00
C01499=1463.793,-178.279,-524.317,180.00,-0.00,180.00
C01500=1471.559,-181.872,-524.297,180.00,0.00,180.00
C01501=1479.662,-184.602,-524.276,180.00,0.00,180.00
C01502=1488.021,-186.442,-524.255,180.00,0.00,180.00
C01503=1496.519,-187.367,-524.234,180.00,0.00,-180.00
C01504=1505.075,-187.367,-524.214,180.00,-0.00,-180.00
C01505=1513.573,-186.442,-524.193,180.00,0.00,180.00
C01506=1521.932,-184.602,-524.172,180.00,0.00,-180.00
C01507=1530.035,-181.872,-524.152,180.00,-0.00,-180.00
C01508=1537.801,-178.279,-524.131,180.00,0.00,180.00
C01509=1545.134,-173.867,-524.110,180.00,0.00,-180.00
C01510=1551.937,-168.696,-524.090,180.00,-0.00,-180.00
C01511=1558.154,-162.807,-524.069,180.00,0.00,180.00
C01512=1563.684,-156.296,-524.048,180.00,0.00,180.00
C01513=1568.487,-149.212,-524.028,180.00,-0.00,-180.00
C01514=1572.495,-141.652,-524.007,180.00,-0.00,-180.00
C01515=1575.658,-133.713,-523.986,180.00,-0.00,180.00
C01516=1577.949,-125.463,-523.966,180.00,-0.00,180.00
C01517=1579.332,-117.028,-523.945,180.00,0.00,180.00
C01518=1579.795,-108.484,-523.924,180.00,0.00,-180.00
C01519=1579.332,-99.940,-523.903,180.00,0.00,-180.00
C01520=1577.949,-91.505,-523.883,180.00,-0.00,-180.00
C01521=1575.658,-83.255,-523.862,180.00,0.00,-180.00
C01522=1572.495,-75.316,-523.841,180.00,-0.00,-180.00
C01523=1568.487,-67.756,-523.821,180.00,-0.00,180.00
C01524=1563.684,-60.672,-523.800,180.00,0.00,-180.00
C01525=1558.154,-54.161,-523.779,180.00,0.00,180.00
C01526=1551.937,-48.272,-523.759,180.00,-0.00,-180.00
C01527=1545.134,-43.101,-523.738,180.00,-0.00,-180.00
C01528=1537.801,-38.689,-523.717,180.00,-0.00,-180.00
C01529=1530.035,-35.096,-523.697,180.00,0.00,-180.00
C01530=1521.932,-32.366,-523.676,180.00,0.00,180.00
C01531=1513.573,-30.526,-523.655,180.00,-0.00,-180.00
C01532=1505.075,-29.601,-523.634,180.00,0.00,-180.00
C01533=1496.519,-29.601,-523.614,180.00,-0.00,-180.00
C01534=1488.021,-30.526,-523.593,180.00,-0.00,-180.00
C01535=1479.662,-32.366,-523.572,180.00,-0.00,-180.00
C01536=1471.559,-35.096,-523.552,180.00,-0.00,-180.00
C01537=1463.793,-38.689,-523.531,180.00,-0.00,-180.00
C01538=1456.460,-43.101,-523.510,180.00,-0.00,-180.00
C01539=1449.657,-48.272,-523.490,180.00,0.00,-180.00
C01540=1443.440,-54.161,-523.469,180.00,-0.00,-180.00
C01541=1437.910,-60.672,-523.448,180.00,0.00,-180.00
C01542=1433.107,-67.756,-523.428,180.00,-0.00,-180.00
C01543=1429.099,-75.316,-523.407,180.00,0.00,-180.00
C01544=1425.936,-83.255,-523.386,180.00,-0.00,180.00
C01545=1423.645,-91.505,-523.366,180.00,-0.00,180.00
C01546=1422.262,-99.940,-523.345,180.00,-0.00,-180.00
C01547=1421.799,-108.484,-523.324,180.00,-0.00,-180.00
C01548=1422.262,-117.028,-523.303,180.00,0.00,180.00
C01549=1423.645,-125.463,-523.283,180.00,-0.00,-180.00
C01550=1425.936,-133.713,-523.262,180.00,0.00,-180.00
C01551=1429.099,-141.652,-523.241,180.00,0.00,-180.00
C01552=1433.107,-149.212,-523.221,180.00,-0.00,-180.00
C01553=1437.910,-156.296,-523.200,180.00,0.00,180.00
C01554=1443.440,-162.807,-523.179,180.00,0.00,-180.00
C01555=1449.657,-168.696,-523.159,180.00,0.00,-180.00
C01556=1456.460,-173.867,-523.138,180.00,0.00,-180.00
C01557=1463.793,-178.279,-523.117,180.00,-0.00,180.00
C01558=1471.559,-181.872,-523.097,180.00,0.00,180.00
C01559=1479.662,-184.602,-523.076,180.00,-0.00,180.00
C01560=1488.021,-186.442,-523.055,180.00,0.00,180.00
C01561=1496.519,-187.367,-523.034,180.00,0.00,-180.00
C01562=1505.075,-187.367,-523.014,180.00,0.00,-180.00
C01563=1513.573,-186.442,-522.993,180.00,-0.00,180.00
C01564=1521.932,-184.602,-522.972,180.00,0.00,-180.00
C01565=1530.035,-181.872,-522.952,180.00,0.00,-180.00
C01566=1537.801,-178.279,-522.931,180.00,-0.00,180.00
C01567=1545.134,-173.867,-522.910,180.00,0.00,-180.00
C01568=1551.937,-168.696,-522.890,180.00,0.00,-180.00
C01569=1558.154,-162.807,-522.869,180.00,0.00,180.00
C01570=1563.684,-156.296,-522.848,180.00,-0.00,180.00
C01571=1568.487,-149.212,-522.828,180.00,0.00,-180.00
C01572=1572.495,-141.652,-522.807,180.00,0.00,-180.00
C01573=1575.658,-133.713,-522.786,180.00,0.00,180.00
C01574=1577.949,-125.463,-522.766,180.00,0.00,180.00
C01575=1579.332,-117.028,-522.745,180.00,0.00,180.00
C01576=1579.795,-108.484,-522.724,180.00,0.00,-180.00
C01577=1579.332,-99.940,-522.703,180.00,-0.00,-180.00
C01578=1577.949,-91.505,-522.683,180.00,0.00,-180.00
C01579=1575.658,-83.255,-522.662,180.00,-0.00,-180.00
C01580=1572.495,-75.316,-522.641,180.00,0.00,-180.00
C01581=1568.487,-67.756,-522.621,180.00,0.00,180.00
C01582=1563.684,-60.672,-522.600,180.00,-0.00,-180.00
C01583=1558.154,-54.161,-522.579,180.00,0.00,180.00
C01584=1551.937,-48.272,-522.559,180.00,0.00,-180.00
C01585=1545.134,-43.101,-522.538,180.00,-0.00,-180.00
C01586=1537.801,-38.689,-522.517,180.00,0.00,-180.00
C01587=1530.035,-35.096,-522.497,180.00,0.00,-180.00
C01588=1521.932,-32.366,-522.476,180.00,0.00,180.00
C01589=1513.573,-30.526,-522.455,180.00,-0.00,-180.00
C01590=1505.075,-29.601,-522.434,180.00,0.00,-180.00
C01591=1496.519,-29.601,-522.414,180.00,0.00,-180.00
C01592=1488.021,-30.526,-522.393,180.00,0.00,-180.00
C01593=1479.662,-32.366,-522.372,180.00,0.00,-180.00
C01594=1471.559,-35.096,-522.352,180.00,-0.00,-180.00
C01595=1463.793,-38.689,-522.331,180.00,0.00,-180.00
C01596=1456.460,-43.101,-522.310,180.00,0.00,-180.00
C01597=1449.657,-48.272,-522.290,180.00,0.00,-180.00
C01598=1443.440,-54.161,-522.269,180.00,0.00,-180.00
C01599=1437.910,-60.672,-522.248,180.00,-0.00,-180.00
C01600=1433.107,-67.756,-522.228,180.00,-0.00,-180.00
C01601=1429.099,-75.316,-522.207,180.00,-0.00,-180.00
C01602=1425.936,-83.255,-522.186,180.00,0.00,180.00
C01603=1423.645,-91.505,-522.166,180.00,0.00,180.00
C01604=1422.262,-99.940,-522.145,180.00,-0.00,-180.00
C01605=1421.799,-108.484,-522.124,180.00,-0.00,-180.00
C01606=1422.262,-117.028,-522.103,180.00,0.00,-180.00
C01607=1423.645,-125.463,-522.083,180.00,0.00,-180.00
C01608=1425.936,-133.713,-522.062,180.00,0.00,-180.00
C01609=1429.099,-141.652,-522.041,180.00,0.00,-180.00
C01610=1433.107,-149.212,-522.021,180.00,-0.00,-180.00
C01611=1437.910,-156.296,-522.000,180.00,0.00,180.00
C01612=1443.440,-162.807,-521.979,180.00,-0.00,-180.00
C01613=1449.657,-168.696,-521.959,180.00,0.00,-180.00
C01614=1456.460,-173.867,-521.938,180.00,-0.00,-180.00
C01615=1463.793,-178.279,-521.917,180.00,0.00,180.00
C01616=1471.559,-181.872,-521.897,180.00,0.00,180.00
C01617=1479.662,-184.602,-521.876,180.00,0.00,180.00
C01618=1488.021,-186.442,-521.855,180.00,0.00,180.00
C01619=1496.519,-187.367,-521.834,180.00,0.00,-180.00
C01620=1505.075,-187.367,-521.814,180.00,0.00,-180.00
C01621=1513.573,-186.442,-521.793,180.00,0.00,180.00
C01622=1521.932,-184.602,-521.772,180.00,0.00,-180.00
C01623=1530.035,-181.872,-521.752,180.00,-0.00,-180.00
C01624=1537.801,-178.279,-521.731,180.00,0.00,180.00
C01625=1545.134,-173.867,-521.710,180.00,0.00,-180.00
C01626=1551.937,-168.696,-521.690,180.00,0.00,-180.00
C01627=1558.154,-162.807,-521.669,180.00,0.00,180.00
C01628=1563.684,-156.296,-521.648,180.00,0.00,180.00
C01629=1568.487,-149.212,-521.628,180.00,0.00,-180.00
C01630=1572.495,-141.652,-521.607,180.00,-0.00,-180.00
C01631=1575.658,-133.713,-521.586,180.00,-0.00,180.00
C01632=1577.949,-125.463,-521.566,180.00,-0.00,180.00
C01633=1579.332,-117.028,-521.545,180.00,0.00,180.00
C01634=1579.795,-108.484,-521.524,180.00,0.00,-180.00
C01635=1579.332,-99.940,-521.503,180.00,-0.00,-180.00
C01636=1577.949,-91.505,-521.483,180.00,-0.00,-180.00
C01637=1575.658,-83.255,-521.462,180.00,0.00,-180.00
C01638=1572.495,-75.316,-521.441,180.00,0.00,-180.00
C01639=1568.487,-67.756,-521.421,180.00,-0.00,180.00
C01640=1563.684,-60.672,-521.400,180.00,0.00,-180.00
C01641=1558.154,-54.161,-521.379,180.00,0.00,180.00
C01642=1551.937,-48.272,-521.359,180.00,0.00,-180.00
C01643=1545.134,-43.101,-521.338,180.00,-0.00,-180.00
C01644=1537.801,-38.689,-521.317,180.00,-0.00,-180.00
C01645=1530.035,-35.096,-521.297,180.00,0.00,-180.00
C01646=1521.932,-32.366,-521.276,180.00,-0.00,180.00
C01647=1513.573,-30.526,-521.255,180.00,0.00,-180.00
C01648=1505.075,-29.601,-521.234,180.00,0.00,-180.00
C01649=1496.519,-29.601,-521.214,180.00,-0.00,-180.00
C01650=1488.021,-30.526,-521.193,180.00,0.00,-180.00
C01651=1479.662,-32.366,-521.172,180.00,-0.00,-180.00
C01652=1471.559,-35.096,-521.152,180.00,-0.00,-180.00
C01653=1463.793,-38.689,-521.131,180.00,-0.00,-180.00
C01654=1456.460,-43.101,-521.110,180.00,0.00,-180.00
C01655=1449.657,-48.272,-521.090,180.00,0.00,-180.00
C01656=1443.440,-54.161,-521.069,180.00,-0.00,-180.00
C01657=1437.910,-60.672,-521.048,180.00,0.00,-180.00
C01658=1433.107,-67.756,-521.028,180.00,-0.00,-180.00
C01659=1429.099,-75.316,-521.007,180.00,0.00,-180.00
C01660=1425.936,-83.255,-520.986,180.00,0.00,180.00
C01661=1423.645,-91.505,-520.966,180.00,-0.00,180.00
C01662=1422.262,-99.940,-520.945,180.00,0.00,-180.00
C01663=1421.799,-108.484,-520.924,180.00,-0.00,-180.00
C01664=1422.262,-117.028,-520.903,180.00,-0.00,-180.00
C01665=1423.645,-125.463,-520.883,180.00,-0.00,-180.00
C01666=1425.936,-133.713,-520.862,180.00,0.00,-180.00
C01667=1429.099,-141.652,-520.841,180.00,0.00,-180.00
C01668=1433.107,-149.212,-520.821,180.00,-0.00,-180.00
C01669=1437.910,-156.296,-520.800,180.00,-0.00,180.00
C01670=1443.440,-162.807,-520.779,180.00,-0.00,-180.00
C01671=1449.657,-168.696,-520.759,180.00,-0.00,-180.00
C01672=1456.460,-173.867,-520.738,180.00,0.00,-180.00
C01673=1463.793,-178.279,-520.717,180.00,0.00,180.00
C01674=1471.559,-181.872,-520.697,180.00,-0.00,180.00
C01675=1479.662,-184.602,-520.676,180.00,0.00,180.00
C01676=1488.021,-186.442,-520.655,180.00,0.00,180.00
C01677=1496.519,-187.367,-520.634,180.00,0.00,-180.00
C01678=1505.075,-187.367,-520.614,180.00,0.00,-180.00
C01679=1513.573,-186.442,-520.593,180.00,0.00,180.00
C01680=1521.932,-184.602,-520.572,180.00,0.00,-180.00
C01681=1530.035,-181.872,-520.552,180.00,-0.00,-180.00
C01682=1537.801,-178.279,-520.531,180.00,0.00,180.00
C01683=1545.134,-173.867,-520.510,180.00,-0.00,-180.00
C01684=1551.937,-168.696,-520.490,180.00,0.00,-180.00
C01685=1558.154,-162.807,-520.469,180.00,0.00,180.00
C01686=1563.684,-156.296,-520.448,180.00,0.00,180.00
C01687=1568.487,-149.212,-520.428,180.00,0.00,-180.00
C01688=1572.495,-141.652,-520.407,180.00,0.00,-180.00
C01689=1575.658,-133.713,-520.386,180.00,0.00,180.00
C01690=1577.949,-125.463,-520.366,180.00,-0.00,180.00
C01691=1579.332,-117.028,-520.345,180.00,0.00,180.00
C01692=1579.795,-108.484,-520.324,180.00,0.00,-180.00
C01693=1579.332,-99.940,-520.303,180.00,0.00,-180.00
C01694=1577.949,-91.505,-520.283,180.00,0.00,-180.00
C01695=1575.658,-83.255,-520.262,180.00,-0.00,-180.00
C01696=1572.495,-75.316,-520.241,180.00,0.00,-180.00
C01697=1568.487,-67.756,-520.221,180.00,0.00,180.00
C01698=1563.684,-60.672,-520.200,180.00,-0.00,-180.00
C01699=1558.154,-54.161,-520.179,180.00,-0.00,180.00
C01700=1551.937,-48.272,-520.159,180.00,-0.00,-180.00
C01701=1545.134,-43.101,-520.138,180.00,0.00,-180.00
C01702=1537.801,-38.689,-520.117,180.00,0.00,-180.00
C01703=1530.035,-35.096,-520.097,180.00,-0.00,-180.00
C01704=1521.932,-32.366,-520.076,180.00,0.00,180.00
C01705=1513.573,-30.526,-520.055,180.00,0.00,-180.00
C01706=1505.075,-29.601,-520.034,180.00,0.00,-180.00
C01707=1496.519,-29.601,-520.014,180.00,0.00,-180.00
C01708=1488.021,-30.526,-519.993,180.00,0.00,-180.00
C01709=1479.662,-32.366,-519.972,180.00,-0.00,-180.00
C01710=1471.559,-35.096,-519.952,180.00,-0.00,-180.00
C01711=1463.793,-38.689,-519.931,180.00,0.00,-180.00
C01712=1456.460,-43.101,-519.910,180.00,-0.00,-180.00
C01713=1449.657,-48.272,-519.890,180.00,-0.00,-180.00
C01714=1443.440,-54.161,-519.869,180.00,-0.00,-180.00
C01715=1437.910,-60.672,-519.848,180.00,0.00,-180.00
C01716=1433.107,-67.756,-519.828,180.00,0.00,-180.00
C01717=1429.099,-75.316,-519.807,180.00,0.00,-180.00
C01718=1425.936,-83.255,-519.786,180.00,0.00,180.00
C01719=1423.645,-91.505,-519.766,180.00,-0.00,180.00
C01720=1422.262,-99.940,-519.745,180.00,0.00,-180.00
C01721=1421.799,-108.484,-519.724,180.00,-0.00,-180.00
C01722=1422.262,-117.028,-519.703,180.00,0.00,-180.00
C01723=1423.645,-125.463,-519.683,180.00,-0.00,-180.00
C01724=1425.936,-133.713,-519.662,180.00,0.00,-180.00
C01725=1429.099,-141.652,-519.641,180.00,0.00,-180.00
C01726=1433.107,-149.212,-519.621,180.00,-0.00,-180.00
C01727=1437.910,-156.296,-519.600,180.00,0.00,180.00
C01728=1443.440,-162.807,-519.579,180.00,-0.00,-180.00
C01729=1449.657,-168.696,-519.559,180.00,-0.00,-180.00
C01730=1456.460,-173.867,-519.538,180.00,-0.00,-180.00
C01731=1463.793,-178.279,-519.517,180.00,-0.00,180.00
C01732=1471.559,-181.872,-519.497,180.00,-0.00,180.00
C01733=1479.662,-184.602,-519.476,180.00,0.00,180.00
C01734=1488.021,-186.442,-519.455,180.00,0.00,180.00
C01735=1496.519,-187.367,-519.434,180.00,-0.00,-180.00
C01736=1505.075,-187.367,-519.414,180.00,-0.00,-180.00
C01737=1513.573,-186.442,-519.393,180.00,-0.00,180.00
C01738=1521.932,-184.602,-519.372,180.00,0.00,-180.00
C01739=1530.035,-181.872,-519.352,180.00,0.00,-180.00
C01740=1537.801,-178.279,-519.331,180.00,-0.00,180.00
C01741=1545.134,-173.867,-519.310,180.00,0.00,-180.00
C01742=1551.937,-168.696,-519.290,180.00,0.00,-180.00
C01743=1558.154,-162.807,-519.269,180.00,0.00,180.00
C01744=1563.684,-156.296,-519.248,180.00,-0.00,180.00
C01745=1568.487,-149.212,-519.228,180.00,-0.00,-180.00
C01746=1572.495,-141.652,-519.207,180.00,0.00,-180.00
C01747=1575.658,-133.713,-519.186,180.00,-0.00,180.00
C01748=1577.949,-125.463,-519.166,180.00,-0.00,180.00
C01749=1579.332,-117.028,-519.145,180.00,-0.00,180.00
C01750=1579.795,-108.484,-519.124,180.00,0.00,-180.00
C01751=1579.332,-99.940,-519.103,180.00,-0.00,-180.00
C01752=1577.949,-91.505,-519.083,180.00,0.00,-180.00
C01753=1575.658,-83.255,-519.062,180.00,-0.00,-180.00
C01754=1572.495,-75.316,-519.041,180.00,0.00,-180.00
C01755=1568.487,-67.756,-519.021,180.00,0.00,180.00
C01756=1563.684,-60.672,-519.000,180.00,-0.00,-180.00
C01757=1558.154,-54.161,-518.979,180.00,0.00,180.00
C01758=1551.937,-48.272,-518.959,180.00,0.00,-180.00
C01759=1545.134,-43.101,-518.938,180.00,0.00,-180.00
C01760=1537.801,-38.689,-518.917,180.00,-0.00,-180.00
C01761=1530.035,-35.096,-518.897,180.00,-0.00,-180.00
C01762=1521.932,-32.366,-518.876,180.00,0.00,180.00
C01763=1513.573,-30.526,-518.855,180.00,0.00,-180.00
C01764=1505.075,-29.601,-518.834,180.00,-0.00,-180.00
C01765=1496.519,-29.601,-518.814,180.00,0.00,-180.00
C01766=1488.021,-30.526,-518.793,180.00,0.00,-180.00
C01767=1479.662,-32.366,-518.772,180.00,0.00,-180.00
C01768=1471.559,-35.096,-518.752,180.00,0.00,-180.00
C01769=1463.793,-38.689,-518.731,180.00,-0.00,-180.00
C01770=1456.460,-43.101,-518.710,180.00,0.00,-180.00
C01771=1449.657,-48.272,-518.690,180.00,-0.00,-180.00
C01772=1443.440,-54.161,-518.669,180.00,-0.00,-180.00
C01773=1437.910,-60.672,-518.648,180.00,-0.00,-180.00
C01774=1433.107,-67.756,-518.628,180.00,-0.00,-180.00
C01775=1429.099,-75.316,-518.607,180.00,0.00,-180.00
C01776=1425.936,-83.255,-518.586,180.00,0.00,180.00
C01777=1423.645,-91.505,-518.566,180.00,0.00,180.00
C01778=1422.262,-99.940,-518.545,180.00,0.00,-180.00
C01779=1421.799,-108.484,-518.524,180.00,0.00,-180.00
C01780=1422.262,-117.028,-518.503,180.00,-0.00,-180.00
C01781=1423.645,-125.463,-518.483,180.00,-0.00,-180.00
C01782=1425.936,-133.713,-518.462,180.00,0.00,-180.00
C01783=1429.099,-141.652,-518.441,180.00,-0.00,-180.00
C01784=1433.107,-149.212,-518.421,180.00,0.00,-180.00
C01785=1437.910,-156.296,-518.400,180.00,0.00,180.00
C01786=1443.440,-162.807,-518.379,180.00,0.00,-180.00
C01787=1449.657,-168.696,-518.359,180.00,-0.00,-180.00
C01788=1456.460,-173.867,-518.338,180.00,0.00,-180.00
C01789=1463.793,-178.279,-518.317,180.00,0.00,180.00
C01790=1471.559,-181.872,-518.297,180.00,0.00,180.00
C01791=1479.662,-184.602,-518.276,180.00,0.00,180.00
C01792=1488.021,-186.442,-518.255,180.00,0.00,180.00
C01793=1496.519,-187.367,-518.234,180.00,0.00,-180.00
C01794=1505.075,-187.367,-518.214,180.00,-0.00,180.00
C01795=1513.573,-186.442,-518.193,180.00,0.00,180.00
C01796=1521.932,-184.602,-518.172,180.00,0.00,-180.00
C01797=1530.035,-181.872,-518.152,180.00,-0.00,-180.00
C01798=1537.801,-178.279,-518.131,180.00,0.00,180.00
C01799=1545.134,-173.867,-518.110,180.00,0.00,-180.00
C01800=1551.937,-168.696,-518.090,180.00,-0.00,-180.00
C01801=1558.154,-162.807,-518.069,180.00,-0.00,180.00
C01802=1563.684,-156.296,-518.048,180.00,0.00,180.00
C01803=1568.487,-149.212,-518.028,180.00,0.00,-180.00
C01804=1572.495,-141.652,-518.007,180.00,0.00,-180.00
C01805=1575.658,-133.713,-517.986,180.00,0.00,180.00
C01806=1577.949,-125.463,-517.966,180.00,0.00,180.00
C01807=1579.332,-117.028,-517.945,180.00,-0.00,180.00
C01808=1579.795,-108.484,-517.924,180.00,0.00,-180.00
C01809=1579.332,-99.940,-517.903,180.00,0.00,-180.00
C01810=1577.949,-91.505,-517.883,180.00,0.00,-180.00
C01811=1575.658,-83.255,-517.862,180.00,0.00,-180.00
C01812=1572.495,-75.316,-517.841,180.00,-0.00,-180.00
C01813=1568.487,-67.756,-517.821,180.00,0.00,180.00
C01814=1563.684,-60.672,-517.800,180.00,0.00,-180.00
C01815=1558.154,-54.161,-517.779,180.00,0.00,180.00
C01816=1551.937,-48.272,-517.759,180.00,0.00,-180.00
C01817=1545.134,-43.101,-517.738,180.00,-0.00,-180.00
C01818=1537.801,-38.689,-517.717,180.00,0.00,-180.00
C01819=1530.035,-35.096,-517.697,180.00,-0.00,-180.00
C01820=1521.932,-32.366,-517.676,180.00,-0.00,180.00
C01821=1513.573,-30.526,-517.655,180.00,0.00,-180.00
C01822=1505.075,-29.601,-517.634,180.00,-0.00,-180.00
C01823=1496.519,-29.601,-517.614,180.00,0.00,-180.00
C01824=1488.021,-30.526,-517.593,180.00,-0.00,-180.00
C01825=1479.662,-32.366,-517.572,180.00,0.00,-180.00
C01826=1471.559,-35.096,-517.552,180.00,0.00,-180.00
C01827=1463.793,-38.689,-517.531,180.00,0.00,-180.00
C01828=1456.460,-43.101,-517.510,180.00,0.00,-180.00
C01829=1449.657,-48.272,-517.490,180.00,0.00,-180.00
C01830=1443.440,-54.161,-517.469,180.00,0.00,-180.00
C01831=1437.910,-60.672,-517.448,180.00,-0.00,-180.00
C01832=1433.107,-67.756,-517.428,180.00,0.00,-180.00
C01833=1429.099,-75.316,-517.407,180.00,0.00,-180.00
C01834=1425.936,-83.255,-517.386,180.00,-0.00,180.00
C01835=1423.645,-91.505,-517.366,180.00,0.00,180.00
C01836=1422.262,-99.940,-517.345,180.00,-0.00,-180.00
C01837=1421.799,-108.484,-517.324,180.00,-0.00,-180.00
C01838=1422.262,-117.028,-517.303,180.00,-0.00,-180.00
C01839=1423.645,-125.463,-517.283,180.00,0.00,-180.00
C01840=1425.936,-133.713,-517.262,180.00,0.00,-180.00
C01841=1429.099,-141.652,-517.241,180.00,0.00,-180.00
C01842=1433.107,-149.212,-517.221,180.00,0.00,-180.00
C01843=1437.910,-156.296,-517.200,180.00,-0.00,180.00
C01844=1443.440,-162.807,-517.179,180.00,-0.00,-180.00
C01845=1449.657,-168.696,-517.159,180.00,0.00,-180.00
C01846=1456.460,-173.867,-517.138,180.00,0.00,-180.00
C01847=1463.793,-178.279,-517.117,180.00,0.00,180.00
C01848=1471.559,-181.872,-517.097,180.00,0.00,180.00
C01849=1479.662,-184.602,-517.076,180.00,0.00,180.00
C01850=1488.021,-186.442,-517.055,180.00,0.00,180.00
C01851=1496.519,-187.367,-517.034,180.00,-0.00,-180.00
C01852=1505.075,-187.367,-517.014,180.00,0.00,180.00
C01853=1513.573,-186.442,-516.993,180.00,0.00,180.00
C01854=1521.932,-184.602,-516.972,180.00,-0.00,-180.00
C01855=1530.035,-181.872,-516.952,180.00,0.00,-180.00
C01856=1537.801,-178.279,-516.931,180.00,-0.00,180.00
